(* Call ST08_404_Y52_0 Hub Bandstrecke STN8 AST (Valve) *)
Analyze         (InputExp:=  TRUE,
                 DoAnalyze:= TRUE );
ST08_404_Y52_0.strAnlayse:=Analyze.OutString;
ST08_404_Y52_0                 (Enable  :=  Analyze.ExpResult,
                                sVisu:=Visu.ST08_404_Y52_0,
                                Reset:=gResetAll,
);
ST08_406_B54_1(ValveObject:= ADR(ST08_404_Y52_0));(*Hub Bandstrecke AST*)
ST08_406_B54_2(ValveObject:= ADR(ST08_404_Y52_0));(*Hub Bandstrecke AST*)

(* Rüstsatz Förderband Vereinzelner (Valve) *)
Analyze         (InputExp:=  TRUE,
                 DoAnalyze:= TRUE );
ST08_412_Y55_0.strAnlayse:=Analyze.OutString;
ST08_412_Y55_0                 (Enable  :=  Analyze.ExpResult,
                                sVisu:=Visu.ST08_412_Y55_0,
                                Reset:=gResetAll,
);

ST08_412_B58_0(ValveObject:= ADR(ST08_412_Y55_0));(*ST08_412_B58_0 Rüstsatz Förderband Vereinzelner eingefahren*)
ST08_412_B58_1(ValveObject:= ADR(ST08_412_Y55_0));(*ST08_412_B58_1 Rüstsatz Förderband Vereinzelner ausgefahren*)

(* Rüstsatz Förderband Stopper (Valve) *)
Analyze         (InputExp:=  TRUE,
                 DoAnalyze:= TRUE );
ST08_412_Y55_2.strAnlayse:=Analyze.OutString;
ST08_412_Y55_2                 (Enable  :=  Analyze.ExpResult,
                                sVisu:=Visu.ST08_412_Y55_2,
                                Reset:=gResetAll,
);

ST08_412_B58_2(ValveObject:= ADR(ST08_412_Y55_2));(*ST08_412_B58_2 Rüstsatz Förderband Stopper eingefahren*)
ST08_412_B58_3(ValveObject:= ADR(ST08_412_Y55_2));(*ST08_412_B58_3 Rüstsatz Förderband Stopper ausgefahren*)
END_PROGRAM

(* POU Stations/ST_00/ST00_SFCs/_CallSFCs, ST *)
PROGRAM _CallSFCs
VAR
	b_init							:BOOL:=FALSE;
	FBSocketCloseAll		:FB_SocketCloseAll;

END_VAR
IF	NOT b_init THEN
		FBSocketCloseAll(bExecute:=TRUE);
		IF	FBSocketCloseAll.bBusy THEN
			b_init:=TRUE;
		END_IF
ELSE
	FBSocketCloseAll(bExecute:=FALSE);
END_IF



ST00_CallSFCs();
ST02_CallSFCs();
ST03_CallSFCs();
ST08_CallSFCs();
END_PROGRAM

(* POU Stations/ST_00/ST00_SFCs/ST00_CallSFCs, ST *)
PROGRAM ST00_CallSFCs
VAR

END_VAR
CallSpecialModeSFCs();

HomePositionSFC();
(*ST00_LoadTInfo();*)
ST02_HomePosition();
ST03_HomePosition();
ST08_HomePosition();
END_PROGRAM

(* POU Stations/ST_02_RT_Tampondrucker/ST02_SFCs/ST02_CallSFCs, ST *)
PROGRAM ST02_CallSFCs

VAR
	fb_ton_wz	:TON;
END_VAR
fb_ton_wz(IN:= TRUE, PT:= t#30s , Q=> , ET=> );

(*Aufrufe nur wenn ein Tampondrucker angeschlossen ist, sonst kommen viele Fehlermeldungt*)
IF	gTypeCode=4991 OR		(*102pol*)
	gTypeCode=312	THEN	(*93pol*)
	ST02_Main();
	ST02_Main.FB_CurrentStepHistorie(st_CurrentStep:=ST02_Main.SFCCurrentStep);
	ST02_AutoStop();
	ST02_CallFBs();
END_IF
(*Sonst werden die Visuelemente nicht mit Texten befüllt*)
IF	ModeSelect.Mode<=MODE_MANUAL AND
	NOT fb_ton_wz.Q THEN
	ST02_CallFBs();
END_IF

	(*Sensopart Kamera initialisieren*)
IF 	NOT MP.ST02.SensopartEthernet THEN
	IF NOT ST02_DT_95_A1.b_ready THEN
		ST02_DT_95_A1.b_init := TRUE;
	ELSE
		ST02_DT_95_A1.b_init := FALSE;
	END_IF
ELSE
	(*Sensopart Kamera Ethernet initialisieren*)
	IF NOT ST02_DT_95_A2.st_ctrl_out.b_bereit AND MP.ST02.SensopartIPAdress <>''  THEN
		ST02_DT_95_A2.st_ctrl_in.b_init := TRUE;
	ELSE
		ST02_DT_95_A2.st_ctrl_in.b_init := FALSE;
	END_IF
END_IF
END_PROGRAM

(* POU Stations/ST_02_RT_Tampondrucker/ST02_FBs/ST02_CallFBs, ST *)
PROGRAM ST02_CallFBs
VAR

END_VAR
(*----------------------------------------------------------------------------------------------------------------------------------*)
(* ----------------------------------------------------------------------------------------- *)
(* Call ST02_FDB_40_B61 Iso von SPM auf Band abgelegt (DigIn) *)
ST02_FDB_40_B61                (sVisu:=Visu.ST02_FDB_40_B61,
                                Reset:=gResetAll,
			(*	CheckSignalHigh:=TRUE,*)
);
(* Call ST02_FDB_40_B71 ST02 Iso auf Band vor Vereinzler (DigIn) *)
ST02_FDB_40_B71                (sVisu:=Visu.ST02_FDB_40_B71,
                                Reset:=gResetAll,
			(*	CheckSignalHigh:=TRUE,*)
);
(* Call ST02_S1_6A01 ST02 Sicherung 24V (DigIn) *)
ST02_S1_6A01                (sVisu:=Visu.ST02_S1_6A01,
                                Reset:=gResetAll,
				CheckSignalHigh:=TRUE,
);

(*Sensopart Kamera für die Erkennung der Markierungen*)
ST02_DT_95_A1(
	b_kamera_aktiv:=MP.ST02.CamOn AND NOT MP.ST02.SensopartEthernet,
	st_Description:= 'Kamera Farberkennung',
	b_reset:=gResetAll );

(*Sensopart Kamera für die Erkennung der Markierungen*)
ST02_DT_95_A2(
	st_ctrl_in := ST02_DT_95_A2.st_ctrl_in,
	Activated := MP.ST02.CamOn AND MP.ST02.SensopartEthernet AND MP.ST02.SensopartIPAdress <> '',
	st_Description:= 'Kamera Farberkennung',
	);
IF 	MP.ST02.SensopartIPAdress <> ''  THEN
	ST02_DT_95_A2.s_IpAdress := MP.ST02.SensopartIPAdress;  		(* 'MP.SensopartIPAdress';*)
	ST02_DT_95_A2.i_CmdPort := 2006;
	ST02_DT_95_A2.i_DataPort :=2005;
END_IF

(* Call ST02_S1_70K61_A1 Start  Bedrucken (DigOutIn) *)
ST02_S1_70K61_A1                  (sVisu:=Visu.ST02_S1_70K61_A1,
                                Reset:=gResetAll,
);

(* Call ST02_62_Y6 Tisch drehen 0 - 180 Grad  (Valve) *)
Analyze         (InputExp:=  TRUE,
                 DoAnalyze:= TRUE );
ST02_62_Y6.strAnlayse:=Analyze.OutString;
ST02_62_Y6                 (Enable  :=  Analyze.ExpResult,
                                sVisu:=Visu.ST02_62_Y6,
                                Reset:=gResetAll,
);
ST02_DT_62_B81(ValveObject:= ADR(ST02_62_Y6));(*Tisch drehen 0 Grad*)
ST02_DT_62_B91(ValveObject:= ADR(ST02_62_Y6));(*Tisch drehen 180 Grad*)

IF	ST02_DT_62_B81.ValveSensor THEN
	MP.ST02.TableData[1].ProcessData.Nest_Nr:=2;
	MP.ST02.TableData[2].ProcessData.Nest_Nr:=1;
ELSIF	ST02_DT_62_B91.ValveSensor THEN
	MP.ST02.TableData[1].ProcessData.Nest_Nr:=1;
	MP.ST02.TableData[2].ProcessData.Nest_Nr:=2;
ELSE
	MP.ST02.TableData[1].ProcessData.Nest_Nr:=0;
	MP.ST02.TableData[2].ProcessData.Nest_Nr:=0;
END_IF
(*----------------------------------------------------------------------------------------------------------------------------------*)
(* Call ST02_62_Y9 Schwenkarm 2 drehen 90 - 180 Grad  (Valve) *)
Analyze         (InputExp:=  TRUE,
                 DoAnalyze:= TRUE );
ST02_62_Y9.strAnlayse:=Analyze.OutString;
ST02_62_Y9                 (Enable  :=  Analyze.ExpResult,
                                sVisu:=Visu.ST02_62_Y9,
                                Reset:=gResetAll,
);
(*ST02_DT_61_B21(ValveObject:= ADR(ST02_62_Y9));		(*Schwenkarm 2 90 Grad*)*)
ST02_DT_61_B11(ValveObject:= ADR(ST02_62_Y9));		(*Schwenkarm 2 180 Grad*)

(* Call ST02_62_Y11 Schwenkarm 2 drehen 90 - 0 Grad  (Valve) *)
Analyze         (InputExp:=  TRUE,
                 DoAnalyze:= TRUE );
ST02_62_Y11.strAnlayse:=Analyze.OutString;
ST02_62_Y11                 (Enable  :=  Analyze.ExpResult,
                                sVisu:=Visu.ST02_62_Y11,
                                Reset:=gResetAll,
);
(*ST02_DT_61_B21_clone(ValveObject:= ADR(ST02_62_Y11));(*Schwenkarm 2 90 Grad*)*)
ST02_DT_61_B31(ValveObject:= ADR(ST02_62_Y11));		(*Schwenkarm 2 0 Grad*)


ST02_Schwenkarm[2](
	ST02_90_180:=ST02_62_Y9 ,
	ST02_90_0:=ST02_62_Y11 ,
	ST02_90:=ST02_DT_61_B21);
(*----------------------------------------------------------------------------------------------------------------------------------*)
(* Call ST02_62_Y13 Schwenkarm 1 drehen 90 - 180 Grad  (Valve) *)
Analyze         (InputExp:=  TRUE,
                 DoAnalyze:= TRUE );
ST02_62_Y13.strAnlayse:=Analyze.OutString;
ST02_62_Y13                 (Enable  :=  Analyze.ExpResult,
                                sVisu:=Visu.ST02_62_Y13,
                                Reset:=gResetAll,
);
(*ST02_DT_61_B51(ValveObject:= ADR(ST02_62_Y13));		(*Schwenkarm 1 90 Grad*)*)
ST02_DT_61_B41(ValveObject:= ADR(ST02_62_Y13));		(*Schwenkarm 1 180 Grad*)

(* Call ST02_62_Y15 Schwenkarm 1 drehen 90 - 0 Grad  (Valve) *)
Analyze         (InputExp:=  TRUE,
                 DoAnalyze:= TRUE );
ST02_62_Y15.strAnlayse:=Analyze.OutString;
ST02_62_Y15                 (Enable  :=  Analyze.ExpResult,
                                sVisu:=Visu.ST02_62_Y15,
                                Reset:=gResetAll,
);
(*ST02_DT_61_B51_clone(ValveObject:= ADR(ST02_62_Y15));(*Schwenkarm 1 90 Grad*)*)
ST02_DT_62_B11(ValveObject:= ADR(ST02_62_Y15));		(*Schwenkarm 1 0 Grad*)

ST02_Schwenkarm[1](
	ST02_90_180:=ST02_62_Y13 ,
	ST02_90_0:=ST02_62_Y15,
	ST02_90:=ST02_DT_61_B51);

(* Call ST02_S1_40K01  Freigabe Förderband von SPM (DigIn) *)
ST02_S1_40K01                     (sVisu:=Visu.ST02_S1_40K01,
                                Reset:=gResetAll,
																CheckSignalHigh:=FALSE,
);
(* Call ST02_FDB_80_B02 Band Entnahmeposition 2 (DigIn) *)
ST02_FDB_80_B02                     (sVisu:=Visu.ST02_FDB_80_B02,
                                Reset:=gResetAll
);

(* Call ST02_FDB_54_B41 Kamera ISK anwesend an Prüfposition (DigIn) *)
ST02_FDB_54_B41               (sVisu:=Visu.ST02_FDB_54_B41,
                                Reset:=gResetAll,
);

(* Call ST02_DT_65B11 Tampondrucker Nest 1 leer (DigIn) *)
ST02_DT_65B11               (sVisu:=Visu.ST02_DT_65B11,
                                Reset:=gResetAll,
);

(* Call ST02_DT_65B21 Tampondrucker Nest 2 leer (DigIn) *)
ST02_DT_65B21               (sVisu:=Visu.ST02_DT_65B21,
                                Reset:=gResetAll,
);
(* Init ST02_35_S31 ST02 Druckschalter Wartungseinheit Hauptluft min.6 bar (DigIn) *)
ST02_35_S31 	                (sVisu:=Visu.ST02_35_S31,
                                Reset:=gResetAll,
			CheckSignalHigh:=TRUE,
);
(*----------------------------------------------------------------------------------------------------------------------------------*)
(* Call ST02_FDB_55X1_5_READY IFM Kamera Flügelerkennung links Ready (DigIn) *)
ST02_FDB_55X1_5_READY               (sVisu:=Visu.ST02_FDB_55X1_5_READY,
                                Reset:=gResetAll,
);
(* Call ST02_FDB_55X1_6_IO IFM Kamera Flügelerkennung links Ergebnis iO (DigIn) *)
ST02_FDB_55X1_6_IO               (sVisu:=Visu.ST02_FDB_55X1_6_IO,
                                Reset:=gResetAll,
);
(* Call ST02_FDB_55X1_6_NIO IFM Kamera Flügelerkennung links Ergebnis niO (DigIn) *)
ST02_FDB_55X1_6_NIO               (sVisu:=Visu.ST02_FDB_55X1_6_NIO,
                                Reset:=gResetAll,
);
(* Call ST02_FDB_55X1_2_TRIGGER IFM Kamera Flügelerkennung links Trigger (DigOutIn) *)
ST02_FDB_55X1_2_TRIGGER                  (sVisu:=Visu.ST02_FDB_55X1_2_TRIGGER,
                                Reset:=gResetAll,
);
(* Call ST02_FDB_55X1_7_JOB_BIT1 IFM Kamera  links Jobwechsel Bit1 (DigOutIn) *)
ST02_FDB_55X1_7_JOB_BIT1                  (sVisu:=Visu.ST02_FDB_55X1_7_JOB_BIT1,
                                Reset:=gResetAll,
);
(* Call ST02_FDB_55X1_7_JOB_BIT2 IFM Kamera  links Jobwechsel Bit2 (DigOutIn) *)
ST02_FDB_55X1_7_JOB_BIT2                  (sVisu:=Visu.ST02_FDB_55X1_7_JOB_BIT2,
                                Reset:=gResetAll,
);
(* Call ST02_FDB_56X1_5_READY IFM Kamera Flügelerkennung rechts Ready (DigIn) *)
ST02_FDB_56X1_5_READY               (sVisu:=Visu.ST02_FDB_56X1_5_READY,
                                Reset:=gResetAll,
);
(* Call ST02_FDB_56X1_6_IO IFM Kamera Flügelerkennung rechts Ergebnis iO (DigIn) *)
ST02_FDB_56X1_6_IO               (sVisu:=Visu.ST02_FDB_56X1_6_IO,
                                Reset:=gResetAll,
);
(* Call ST02_FDB_56X1_6_NIO IFM Kamera Flügelerkennung rechts Ergebnis niO (DigIn) *)
ST02_FDB_56X1_6_NIO               (sVisu:=Visu.ST02_FDB_56X1_6_NIO,
                                Reset:=gResetAll,
);
(* Call ST02_FDB_56X1_2_TRIGGER IFM Kamera Flügelerkennung rechts Trigger (DigOutIn) *)
ST02_FDB_56X1_2_TRIGGER                  (sVisu:=Visu.ST02_FDB_56X1_2_TRIGGER,
                                Reset:=gResetAll,
);
(* Call ST02_FDB_56X1_7_JOB_BIT1 IFM Kamera  rechts Jobwechsel Bit1 (DigOutIn) *)
ST02_FDB_56X1_7_JOB_BIT1                  (sVisu:=Visu.ST02_FDB_56X1_7_JOB_BIT1,
                                Reset:=gResetAll,
);
(* Call ST02_FDB_56X1_7_JOB_BIT2 IFM Kamera  rechts Jobwechsel Bit2 (DigOutIn) *)
ST02_FDB_56X1_7_JOB_BIT2                  (sVisu:=Visu.ST02_FDB_56X1_7_JOB_BIT2,
                                Reset:=gResetAll,
);
(* Call ST02_62_Y4 Kamera Ausschleusen Bandstrecke (Valve) *)
Analyze         (InputExp:=  TRUE,
                 DoAnalyze:= TRUE );
ST02_62_Y4.strAnlayse:=Analyze.OutString;
ST02_62_Y4                 (Enable  :=  Analyze.ExpResult,
                                sVisu:=Visu.ST02_62_Y4,
                                Reset:=gResetAll,
);
ST02_FDB_54_B11(ValveObject:= ADR(ST02_62_Y4));(*Kamera Ausschleusen Bandstrecke eingefahren*)
ST02_FDB_54_B21(ValveObject:= ADR(ST02_62_Y4));(*Kamera Ausschleusen Bandstrecke ausgefahren*)


(*Call ST02_62_Y17 Schwenkarm 1 ISK Fixierung ein/ausfahren(Valve) (Valve) *)
Analyze         (InputExp:=  TRUE,
                 DoAnalyze:= TRUE );
ST02_62_Y17.strAnlayse:=Analyze.OutString;
ST02_62_Y17                 (Enable  :=  Analyze.ExpResult,
                                sVisu:=Visu.ST02_62_Y17,
                                Reset:=gResetAll,
);
ST02_S1_66_B11(ValveObject:= ADR(ST02_62_Y17));(*Kamera Ausschleusen Bandstrecke eingefahren*)
ST02_S1_66_B21(ValveObject:= ADR(ST02_62_Y17));(*Kamera Ausschleusen Bandstrecke ausgefahren*)


(*Call ST02_62_Y18 Schwenkarm 2 ISK Fixierung ein/ausfahren(Valve) (Valve) *)
Analyze         (InputExp:=  TRUE,
                 DoAnalyze:= TRUE );
ST02_62_Y18.strAnlayse:=Analyze.OutString;
ST02_62_Y18                 (Enable  :=  Analyze.ExpResult,
                                sVisu:=Visu.ST02_62_Y18,
                                Reset:=gResetAll,
);
ST02_S1_66_B31(ValveObject:= ADR(ST02_62_Y18));(*Kamera Ausschleusen Bandstrecke eingefahren*)
ST02_S1_66_B41(ValveObject:= ADR(ST02_62_Y18));(*Kamera Ausschleusen Bandstrecke ausgefahren*)


(* Call ST02_35Y01 Einschaltventil Hauptluft Tampondruckanlage (Valve) *)
Analyze         (InputExp:=  TRUE,
                 DoAnalyze:= TRUE );
ST02_35Y01.strAnlayse:=Analyze.OutString;
ST02_35Y01               (Enable  :=  Analyze.ExpResult,
                                sVisu:=Visu.ST02_35Y01,
                                Reset:=gResetAll,
);
END_PROGRAM

(* POU Stations/ST_03_Ruestsaetze/ST_03_FBs/ST03_CallSFCs, ST *)
PROGRAM ST03_CallSFCs


VAR


END_VAR
ST03_Main();
ST03_Main.FB_CurrentStepHistorie(st_CurrentStep:=ST03_Main.SFCCurrentStep);


	(*Sensopart Kamera initialisieren*)
IF NOT MP.ST02.SensopartEthernet THEN
	IF NOT ST03_8_80_A1.b_ready THEN
		ST03_8_80_A1.b_init := TRUE;
	ELSE
		ST03_8_80_A1.b_init := FALSE;
	END_IF
	IF NOT ST03_8_85_A1.b_ready THEN
		ST03_8_85_A1.b_init := TRUE;
	ELSE
		ST03_8_85_A1.b_init := FALSE;
	END_IF
ELSE
	(*Sensopart Kamera Ethernet initialisieren*)
	IF NOT ST03_8_90_A1.st_ctrl_out.b_bereit AND MP.ST02.SensopartIPAdress <>''  THEN
		ST03_8_90_A1.st_ctrl_in.b_init := TRUE;
	ELSE
		ST03_8_90_A1.st_ctrl_in.b_init := FALSE;
	END_IF

	IF NOT ST03_8_95_A1.st_ctrl_out.b_bereit AND MP.ST02.SensopartIPAdress2 <>''  THEN
		ST03_8_95_A1.st_ctrl_in.b_init := TRUE;
	ELSE
		ST03_8_95_A1.st_ctrl_in.b_init := FALSE;
	END_IF

	IF NOT ST03_8_100_A1.st_ctrl_out.b_bereit AND MP.ST03.CamOn[1] THEN
		ST03_8_100_A1.st_ctrl_in.b_init := TRUE;
	ELSE
		ST03_8_100_A1.st_ctrl_in.b_init := FALSE;
	END_IF

	IF NOT ST03_8_103_A1.st_ctrl_out.b_bereit AND MP.ST03.CamOn[2] THEN
		ST03_8_103_A1.st_ctrl_in.b_init := TRUE;
	ELSE
		ST03_8_103_A1.st_ctrl_in.b_init := FALSE;
	END_IF

	(*Keyence Kamera Ethernet initialisieren*)
	IF NOT ST03_8_105_A1.st_ctrl_out.b_bereit AND MP.ST03.CamOn_KYE THEN
		ST03_8_105_A1.st_ctrl_in.b_init := TRUE;
	ELSE
		ST03_8_105_A1.st_ctrl_in.b_init := FALSE;
	END_IF


END_IF
END_PROGRAM

(* POU Stations/ST_08_Palettierer/ST_08_SFCs/ST08_CallSFCs, ST *)
 PROGRAM ST08_CallSFCs


VAR


END_VAR
ST08_Process();
ST08_Process.FB_CurrentStepHistorie(st_CurrentStep:=ST08_Process.SFCCurrentStep);

ST08_VV1_Y50_0();
ST08_VV1_Y50_2();

ST08_Depalletizing();
ST08_Depalletizing.FB_CurrentStepHistorie(st_CurrentStep:=ST08_Depalletizing.SFCCurrentStep);

ST08_Palletizing();
ST08_Palletizing.FB_CurrentStepHistorie(st_CurrentStep:=ST08_Palletizing.SFCCurrentStep);
END_PROGRAM

(* POU Stations/ST_08_Palettierer/ST_08_SFCs/Inlett/ST08_VV1_Y50_0, SFC *)
PROGRAM ST08_VV1_Y50_0				(* Vereinzler vor HQE4 *)

VAR_OUTPUT
	SFCCurrentPOU	: STRING:='ST08_VV1_Y50_0';
	SFCCurrentStep	: STRING:='';
	SFCTime			: DINT;
	State   		: DINT;
	Result  		: DINT;
END_VAR
VAR_INPUT

END_VAR
VAR
	MsgOK			: BOOL;
	MsgCancel		: BOOL;
	SFCRun			: BOOL;
	SFCTimeStart	: TIME;
	Delay			: TON;
	TimeOut			: TON;
	(* Userdefinded area *)

END_VAR
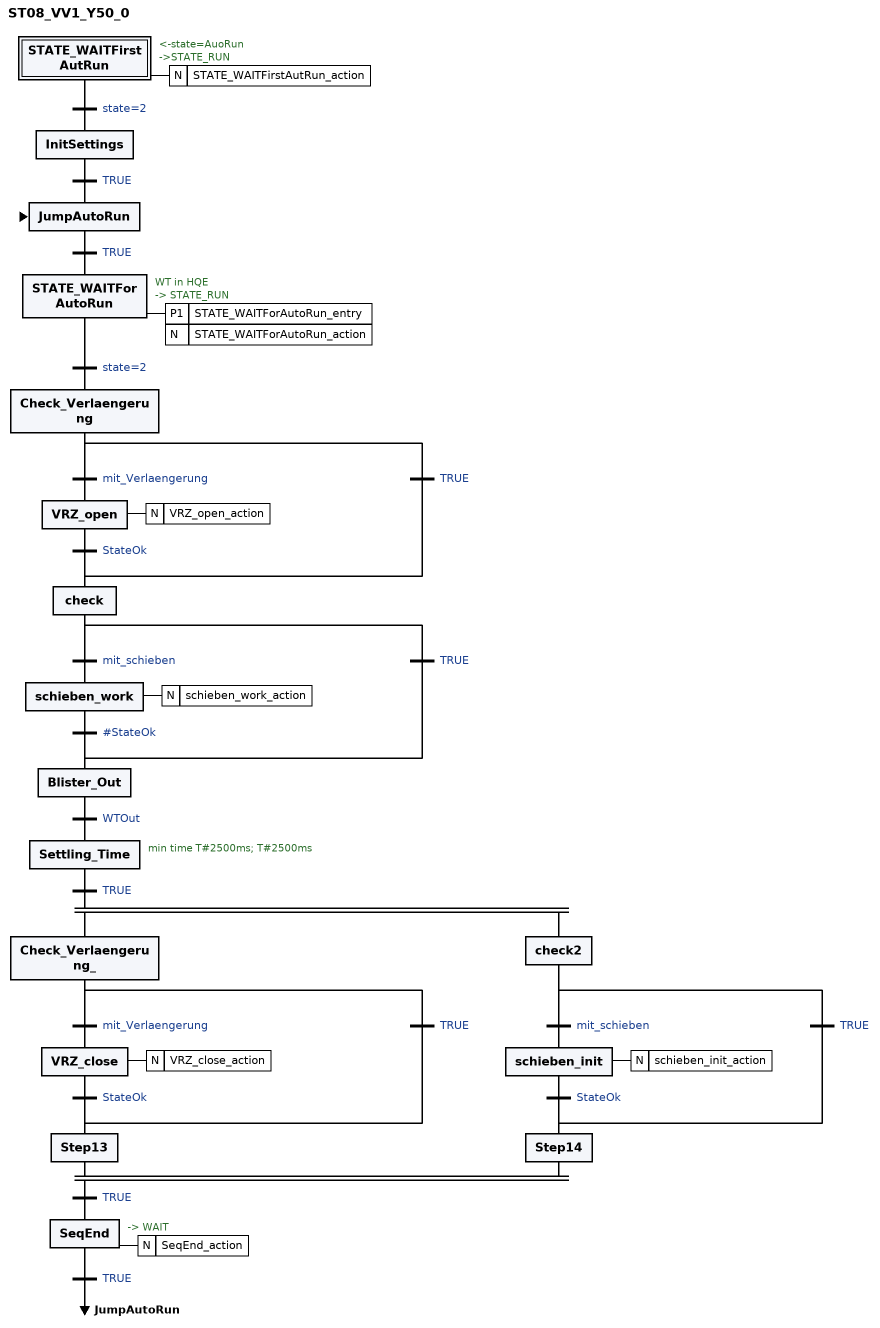
INITIAL_STEP STATE_WAITFirstAutRun: (* <-state=AuoRun / ->STATE_RUN *)
	STATE_WAITFirstAutRun_action(N);
END_STEP
TRANSITION FROM STATE_WAITFirstAutRun TO InitSettings := state=2;
END_TRANSITION
STEP InitSettings:
END_STEP
TRANSITION FROM InitSettings TO JumpAutoRun := TRUE;
END_TRANSITION
STEP JumpAutoRun:
END_STEP
TRANSITION FROM JumpAutoRun TO STATE_WAITForAutoRun := TRUE;
END_TRANSITION
STEP STATE_WAITForAutoRun: (* WT in HQE / -> STATE_RUN *)
	STATE_WAITForAutoRun_entry(P1);
	STATE_WAITForAutoRun_action(N);
END_STEP
TRANSITION FROM STATE_WAITForAutoRun TO Check_Verlaengerung := state=2;
END_TRANSITION
STEP Check_Verlaengerung:
END_STEP
TRANSITION FROM Check_Verlaengerung TO VRZ_open := mit_Verlaengerung;
END_TRANSITION
TRANSITION FROM Check_Verlaengerung TO check := TRUE;
END_TRANSITION
STEP VRZ_open:
	VRZ_open_action(N);
END_STEP
TRANSITION FROM VRZ_open TO check := StateOk;
END_TRANSITION
STEP check:
END_STEP
TRANSITION FROM check TO schieben_work := mit_schieben;
END_TRANSITION
TRANSITION FROM check TO Blister_Out := TRUE;
END_TRANSITION
STEP schieben_work:
	schieben_work_action(N);
END_STEP
TRANSITION FROM schieben_work TO Blister_Out := #StateOk;
END_TRANSITION
STEP Blister_Out:
END_STEP
TRANSITION FROM Blister_Out TO Settling_Time := WTOut;
END_TRANSITION
STEP Settling_Time: (* min time T#2500ms; T#2500ms *)
END_STEP
TRANSITION FROM Settling_Time TO (Check_Verlaengerung_, check2) := TRUE;
END_TRANSITION
STEP Check_Verlaengerung_:
END_STEP
TRANSITION FROM Check_Verlaengerung_ TO VRZ_close := mit_Verlaengerung;
END_TRANSITION
TRANSITION FROM Check_Verlaengerung_ TO Step13 := TRUE;
END_TRANSITION
STEP VRZ_close:
	VRZ_close_action(N);
END_STEP
TRANSITION FROM VRZ_close TO Step13 := StateOk;
END_TRANSITION
STEP Step13:
END_STEP
STEP check2:
END_STEP
TRANSITION FROM check2 TO schieben_init := mit_schieben;
END_TRANSITION
TRANSITION FROM check2 TO Step14 := TRUE;
END_TRANSITION
STEP schieben_init:
	schieben_init_action(N);
END_STEP
TRANSITION FROM schieben_init TO Step14 := StateOk;
END_TRANSITION
STEP Step14:
END_STEP
TRANSITION FROM (Step13, Step14) TO SeqEnd := TRUE;
END_TRANSITION
STEP SeqEnd: (* -> WAIT *)
	SeqEnd_action(N);
END_STEP
TRANSITION FROM SeqEnd TO JumpAutoRun := TRUE;
END_TRANSITION

ACTION STATE_WAITFirstAutRun_action:
IF 		ModeSelect.Mode=MODE_AUTO_RUN
	OR 	ModeSelect.Mode=MODE_STEP_RUN
  OR SpecialMode01.State=State_Run
THEN
	State:=STATE_RUN;
	Result:=RESULT_NON;
ELSE
	State:=STATE_WAIT;
	SFCRun:=FALSE;
(*ELSE*)
END_IF
END_ACTION

ACTION STATE_WAITForAutoRun_entry:
Delay(In:=FALSE);
END_ACTION

ACTION STATE_WAITForAutoRun_action:
Delay(IN:=
	NOT ST08_400_B50_0.BitInToCheck AND
	ST08_401_B50_5.BitInToCheck AND
	ST08_400_Y50_2.InitPosition,
	PT:=T#1500ms);
IF 	((	ModeSelect.Mode=MODE_AUTO_RUN OR 	ModeSelect.Mode=MODE_STEP_RUN   OR SpecialMode01.State=State_Run  )
	AND Delay.Q )

THEN
	State:=STATE_RUN;
	Result:=RESULT_NON;
	SFCTimeStart:=TIME();
ELSE
	State:=STATE_WAIT;
END_IF
END_ACTION

ACTION VRZ_open_action:
ST08_400_Y50_0.MoveWork:=TRUE;
END_ACTION

ACTION schieben_work_action:
ST08_401_Y52_4.MoveWork:=TRUE;
END_ACTION

ACTION VRZ_close_action:
ST08_400_Y50_0.MoveInit:=TRUE;
END_ACTION

ACTION schieben_init_action:
ST08_401_Y52_4.MoveInit:=TRUE;
END_ACTION

ACTION SeqEnd_action:
SFCTime:=TIME_TO_DINT(TIME()-SFCTimeStart);
State:=STATE_WAIT;
END_ACTION

TRANSITION mit_Verlaengerung:
mp.ST08.Trayzufuhr_Verlaengerung
END_TRANSITION

TRANSITION StateOk:
ST08_400_Y50_0.State=STATE_OK
END_TRANSITION

TRANSITION mit_schieben:
MP.ST08.Traystapel_schieben AND
MP.ST08.Trayzufuhr_Verlaengerung
END_TRANSITION

TRANSITION #StateOk:
ST08_401_Y52_4.State=STATE_OK
END_TRANSITION

TRANSITION WTOut:
ST08_400_B50_0.BitInToCheck=TRUE AND ST08_401_B50_5.BitInToCheck=FALSE
END_TRANSITION

TRANSITION mit_Verlaengerung:
MP.ST08.Trayzufuhr_Verlaengerung
END_TRANSITION

TRANSITION StateOk:
ST08_400_Y50_0.State=STATE_OK
END_TRANSITION

TRANSITION mit_schieben:
MP.ST08.Traystapel_schieben AND
MP.ST08.Trayzufuhr_Verlaengerung
END_TRANSITION

TRANSITION StateOk:
ST08_401_Y52_4.State=STATE_OK
END_TRANSITION
END_PROGRAM

(* POU Stations/ST_08_Palettierer/ST_08_SFCs/Inlett/ST08_VV1_Y50_2, SFC *)
PROGRAM ST08_VV1_Y50_2				(* Vereinzler vor HQE4 *)

VAR_OUTPUT
	SFCCurrentPOU	: STRING:='ST08_VV1_Y50_2';
	SFCCurrentStep	: STRING:='';
	SFCTime			: DINT;
	State   		: DINT;
	Result  		: DINT;
END_VAR
VAR_INPUT

END_VAR
VAR
	MsgOK			: BOOL;
	MsgCancel		: BOOL;
	SFCRun			: BOOL;
	SFCTimeStart	: TIME;
	Delay			: TON;
	TimeOut			: TON;
	(* Userdefinded area *)

END_VAR
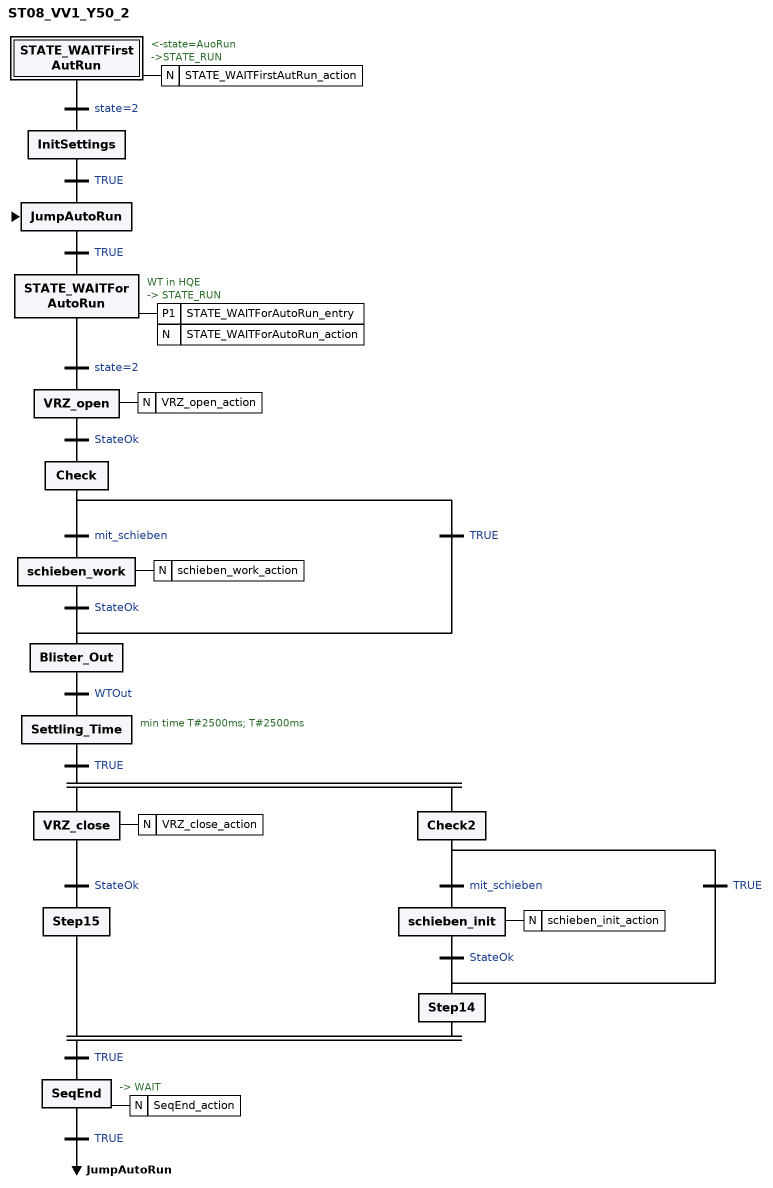
INITIAL_STEP STATE_WAITFirstAutRun: (* <-state=AuoRun / ->STATE_RUN *)
	STATE_WAITFirstAutRun_action(N);
END_STEP
TRANSITION FROM STATE_WAITFirstAutRun TO InitSettings := state=2;
END_TRANSITION
STEP InitSettings:
END_STEP
TRANSITION FROM InitSettings TO JumpAutoRun := TRUE;
END_TRANSITION
STEP JumpAutoRun:
END_STEP
TRANSITION FROM JumpAutoRun TO STATE_WAITForAutoRun := TRUE;
END_TRANSITION
STEP STATE_WAITForAutoRun: (* WT in HQE / -> STATE_RUN *)
	STATE_WAITForAutoRun_entry(P1);
	STATE_WAITForAutoRun_action(N);
END_STEP
TRANSITION FROM STATE_WAITForAutoRun TO VRZ_open := state=2;
END_TRANSITION
STEP VRZ_open:
	VRZ_open_action(N);
END_STEP
TRANSITION FROM VRZ_open TO Check := StateOk;
END_TRANSITION
STEP Check:
END_STEP
TRANSITION FROM Check TO schieben_work := mit_schieben;
END_TRANSITION
TRANSITION FROM Check TO Blister_Out := TRUE;
END_TRANSITION
STEP schieben_work:
	schieben_work_action(N);
END_STEP
TRANSITION FROM schieben_work TO Blister_Out := StateOk;
END_TRANSITION
STEP Blister_Out:
END_STEP
TRANSITION FROM Blister_Out TO Settling_Time := WTOut;
END_TRANSITION
STEP Settling_Time: (* min time T#2500ms; T#2500ms *)
END_STEP
TRANSITION FROM Settling_Time TO (VRZ_close, Check2) := TRUE;
END_TRANSITION
STEP VRZ_close:
	VRZ_close_action(N);
END_STEP
TRANSITION FROM VRZ_close TO Step15 := StateOk;
END_TRANSITION
STEP Step15:
END_STEP
STEP Check2:
END_STEP
TRANSITION FROM Check2 TO schieben_init := mit_schieben;
END_TRANSITION
TRANSITION FROM Check2 TO Step14 := TRUE;
END_TRANSITION
STEP schieben_init:
	schieben_init_action(N);
END_STEP
TRANSITION FROM schieben_init TO Step14 := StateOk;
END_TRANSITION
STEP Step14:
END_STEP
TRANSITION FROM (Step15, Step14) TO SeqEnd := TRUE;
END_TRANSITION
STEP SeqEnd: (* -> WAIT *)
	SeqEnd_action(N);
END_STEP
TRANSITION FROM SeqEnd TO JumpAutoRun := TRUE;
END_TRANSITION

ACTION STATE_WAITFirstAutRun_action:
IF 		ModeSelect.Mode=MODE_AUTO_RUN
	OR 	ModeSelect.Mode=MODE_STEP_RUN
  OR SpecialMode01.State=State_Run
THEN
	State:=STATE_RUN;
	Result:=RESULT_NON;
ELSE
	State:=STATE_WAIT;
	SFCRun:=FALSE;
(*ELSE*)
END_IF
END_ACTION

ACTION STATE_WAITForAutoRun_entry:
Delay(IN:=FALSE);
END_ACTION

ACTION STATE_WAITForAutoRun_action:
Delay(IN:=
	NOT ST08_401_B50_5.BitInToCheck AND
	ST08_402_B51_2.BitInToCheck AND
	ST08_402_Y50_4.InitPosition,
	PT:=T#1500ms);
IF 	((	ModeSelect.Mode=MODE_AUTO_RUN OR 	ModeSelect.Mode=MODE_STEP_RUN   OR SpecialMode01.State=State_Run  )
	AND Delay.Q )

THEN
	State:=STATE_RUN;
	Result:=RESULT_NON;
	SFCTimeStart:=TIME();
ELSE
	State:=STATE_WAIT;
END_IF
END_ACTION

ACTION VRZ_open_action:
ST08_400_Y50_2.MoveWork:=TRUE;
END_ACTION

ACTION schieben_work_action:
ST08_402_Y52_6.MoveWork:=TRUE;
END_ACTION

ACTION VRZ_close_action:
ST08_400_Y50_2.MoveInit:=TRUE;
END_ACTION

ACTION schieben_init_action:
ST08_402_Y52_6.MoveInit:=TRUE;
END_ACTION

ACTION SeqEnd_action:
SFCTime:=TIME_TO_DINT(TIME()-SFCTimeStart);
State:=STATE_WAIT;
END_ACTION

TRANSITION StateOk:
ST08_400_Y50_2.State=STATE_OK
END_TRANSITION

TRANSITION mit_schieben:
MP.ST08.Traystapel_schieben AND
MP.ST08.Trayzufuhr_Verlaengerung
END_TRANSITION

TRANSITION StateOk:
ST08_402_Y52_6.State=STATE_OK
END_TRANSITION

TRANSITION WTOut:
ST08_401_B50_5.BitInToCheck=TRUE AND ST08_402_B51_2.BitInToCheck=FALSE
END_TRANSITION

TRANSITION StateOk:
ST08_400_Y50_2.State=STATE_OK
END_TRANSITION

TRANSITION mit_schieben:
MP.ST08.Traystapel_schieben AND
MP.ST08.Trayzufuhr_Verlaengerung
END_TRANSITION

TRANSITION StateOk:
ST08_402_Y52_6.State=STATE_OK
END_TRANSITION
END_PROGRAM

(* POU Stations/ST_00/ST00_PRGs/_CallPRGs, ST *)
PROGRAM _CallPRGs
VAR
END_VAR
ST00_CallPRGs();
ST02_CallPRGs();
ST03_CallPRGs();
ST08_CallPRGs();
END_PROGRAM

(* POU Stations/ST_00/ST00_PRGs/ST00_CallPRGs, ST *)
PROGRAM ST00_CallPRGs
VAR
	FB_ReadXmlLineConf		: FB_ReadXmlLine;
	sDescription			: STRING;
END_VAR
Lights_and_Lamps();
Safety_Fuses_AirPressure();
JobManagement();
VisuLogger();

IF 	HomePositionSFC.State = STATE_RUN THEN
	ListHomeNOK(InstName:='ST00 ',Description:=sDescription);
END_IF
FB_ReadXmlLineConf(
	Prefix:= 'CONFIG',
	ID:= 'ST00',
	File:= 'CONFIG.xml',
	Text=> sDescription );


IF gInitOk AND ST_Path.Done THEN
	MachineStates();
	ST_Service();
	ST00_ImpExp_MP(
				path:= MP_LocalDriveRoot,
				filename	:=MP_MPExportFilename);
END_IF

(* Schutztüren *)
IF 	ModeSelect.Mode>MODE_MANUAL AND
	ST00_220_S1.BitInToCheck THEN
	ModeSelect.AskForManual:=TRUE;

END_IF

IF	ModeSelect.Mode>MODE_MANUAL THEN
	ST00_220_S1_S31.SetSignalHigh:=TRUE;
	ST00_245_V1.SetSignalHigh:=TRUE;
END_IF

IF 	ModeSelect.Mode<=MODE_MANUAL THEN
	ST00_220_S1_S31.SetSignalLow:=TRUE;
	ST00_245_V1.SetSignalLow:=TRUE;
END_IF

(* Generierung RoboterOffset *)
gRobotOffset :=  TD.RobotOffset;

gTypeCode:=STRING_TO_DINT(DELETE(TD.TypeCode,1,1));
END_PROGRAM

(* POU Stations/ST_00/ST00_PRGs/Lights_and_Lamps, ST *)
PROGRAM Lights_and_Lamps
VAR
	SignalRed			: BOOL;
	SignalOrange		: BOOL;
	SignalGreen			: BOOL;
	SignalBlue			: BOOL;
	SetOrange			: BOOL;
	FP_MachineLight	: R_TRIG;
	FN_MachineLight	: F_TRIG;
	PartLack			: TON;
	TimeOFF			: TON;
	fb_Blinker			: FB_Blinker;
END_VAR
fb_Blinker(b_start:=TRUE, t_taktzeit_on:=t#1s , t_taktzeit_off:=t#1s , b_blinker_out=> );
(* ----------------------------------------------------------------------------------------- *)
(* Ampel  *)
SignalRed	:= ErrorHandler.bOutError ;
SignalOrange	:= MessageHandler.MessageActive OR SetOrange OR ST03_Test_Parts.fb_Blinker.b_blinker_out;;
IF	ModeSelect.Mode=MODE_AUTO_RUN OR ModeSelect.Mode=MODE_STEP_RUN THEN
	SignalGreen	:=TRUE;
ELSIF
	 ModeSelect.Mode=MODE_AUTO_STOP THEN
	SignalGreen	:=fb_Blinker.b_blinker_out;
ELSE
	SignalGreen	:=FALSE;
END_IF
(*SignalGreen	:= ModeSelect.Mode=MODE_AUTO_RUN OR ModeSelect.Mode=MODE_AUTO_STOP OR ModeSelect.Mode=MODE_STEP_RUN;*)
SignalBlue	:= FALSE; (* Parts Missing *)

(* ----------------------------------------------------------------------------------------- *)
PartLack(IN:= FALSE,PT:=T#60s);
IF  	ModeSelect.Mode>MODE_MANUAL AND
	PartLack.Q THEN
	SetOrange:=TRUE;
ELSE
	SetOrange:=FALSE;
END_IF

IF	CurrentVisu <> 'MANUAL_ST00_0' THEN

	(* Ampel Grün *)
	IF 	ST00_350_H1.State=STATE_WAIT AND
		ST00_350_H1.SignalOut <> SignalRed THEN
		ST00_350_H1.SetSignalHigh:= SignalRed;
		ST00_350_H1.SetSignalLow:= NOT SignalRed;
	END_IF;

	(* Ampel Orange *)
	IF 	ST00_350_H2.State=STATE_WAIT AND
		ST00_350_H2.SignalOut <> SignalOrange	THEN
		ST00_350_H2.SetSignalHigh:= SignalOrange;
		ST00_350_H2.SetSignalLow:= NOT SignalOrange;
	END_IF;
	(* Ampel Rot *)
	IF 	ST00_350_H3.State=STATE_WAIT AND
		ST00_350_H3.SignalOut <> SignalGreen THEN
		ST00_350_H3.SetSignalHigh:= SignalGreen;
		ST00_350_H3.SetSignalLow:= NOT SignalGreen;
	END_IF;
	(*Ampel Blau*)
	(*IF 	ST00_350_H4.State=STATE_WAIT AND
		ST00_350_H4.SignalOut <> SignalBlue THEN
		ST00_350_H4.SetSignalHigh:= SignalBlue;
		ST00_350_H4.SetSignalLow:= NOT SignalBlue;
	END_IF*)

(* Bedientaster-Beleuchtungen *)
	(* H3 Reset *)
	IF 	ST00_292_H3_RESET.State=STATE_WAIT AND
		ST00_292_H3_RESET.SignalOut <> SignalRed THEN
		ST00_292_H3_RESET.SetSignalHigh:=SignalRed;
		ST00_292_H3_RESET.SetSignalLow:= NOT SignalRed;
	END_IF;
	(* H2 Start *)
	IF 	ST00_292_H2_Start.State=STATE_WAIT AND
		ST00_292_H2_Start.SignalOut <> SignalGreen 	THEN
		ST00_292_H2_Start.SetSignalHigh:=SignalGreen;
		ST00_292_H2_Start.SetSignalLow:= NOT SignalGreen;
	END_IF

	(* H3 Reset *)
	IF 	ST00_245_V3_RESET.State=STATE_WAIT AND
		ST00_245_V3_RESET.SignalOut <> SignalRed THEN
		ST00_245_V3_RESET.SetSignalHigh:=SignalRed;
		ST00_245_V3_RESET.SetSignalLow:= NOT SignalRed;
	END_IF;
	(* H2 Start *)
	IF 	ST00_245_V2_START.State=STATE_WAIT AND
		ST00_245_V2_START.SignalOut <> SignalGreen 	THEN
		ST00_245_V2_START.SetSignalHigh:=SignalGreen;
		ST00_245_V2_START.SetSignalLow:= NOT SignalGreen;
	END_IF
END_IF

(* Beleuchtung Anlage Ein, wenn Schutz geöffnet*)
(* ----------------------------------------------------------------------------------------- *)

(* Flag Positive - Light on*)
FP_MachineLight(CLK:=NOT gReadyForControlOn );

(* Flag Negative - Light on*)
FN_MachineLight(CLK:=NOT gReadyForControlOn );

TimeOFF(IN:=ST00_31_K1.SignalOut, PT:=t#5m);

IF 	FP_MachineLight.Q THEN
	ST00_31_K1.SetSignalHigh	:= TRUE;
	ST00_31_K1.SetSignalLow	:= FALSE;
END_IF
IF 	FN_MachineLight.Q OR
	TimeOFF.Q THEN
	ST00_31_K1.SetSignalHigh	:= FALSE;
	ST00_31_K1.SetSignalLow	:= TRUE;
END_IF
END_PROGRAM

(* POU zLibrary/ept/Funktionsbausteine/FB_Blinker, ST *)
FUNCTION_BLOCK FB_Blinker
VAR_INPUT
	b_start 		: BOOL;
	t_taktzeit_on	: TIME;
	t_taktzeit_off	: TIME;
END_VAR
VAR_OUTPUT
	b_blinker_out : BOOL;
END_VAR
VAR
	fb_ton		: TON;
END_VAR
fb_ton(IN:=NOT fb_ton.Q AND b_start , PT:=t_taktzeit_off + t_taktzeit_on , Q=> , ET=> );
b_blinker_out:= fb_ton.ET >= t_taktzeit_off;
END_FUNCTION_BLOCK

(* POU Stations/ST_03_Ruestsaetze/ST_03_SFCs/ST03_Test_Parts, ST *)
PROGRAM ST03_Test_Parts
VAR
	FB_Blinker					: FB_Blinker;
END_VAR
(* An der Oberfläche muss bestätigt werden, dass die Prüfteile entnommen worden sind *)
IF 	gTakeTestPartsFinished OR
	ST_CPU.LNG <> CZ THEN
	ST03_Main.TestPartsRemove := FALSE;
END_IF

(* Meldung blinken bis Teile entnommen werden / Blikani okna odeber vzorky do potvrzeni odebrani*)
fb_Blinker(b_start:=ST03_Main.TestPartsRemove , t_taktzeit_on:=t#1s , t_taktzeit_off:=t#1s , b_blinker_out=> );

(*Beim Dummytest 160 polig dürfen die Isos nicht bedruckt werden
	/ Stop Printing at Dummytest 160 pol*)

IF	gTypeCode=322	THEN 	(*160 polig*)
	IF 	NOT DummyTest_160pol THEN
		IF	ST03_8_B76_1.BitInToCheck OR  (* 3621 *)
			ST03_423_B66_0.BitInToCheck THEN (* Rüstsatz 160 polig LS 1 *)
			ST03_PLAN_70V1_1.SetSignalHigh	:= TRUE;		(* Start  Bedrucken Tintenstrahldrucker Frontseite*)
			ST03_PLAN_70V1_1.SetSignalLow	:= FALSE;
		ELSE
			ST03_PLAN_70V1_1.SetSignalHigh	:= FALSE;	(* Start  Bedrucken Tintenstrahldrucker Frontseite*)
			ST03_PLAN_70V1_1.SetSignalLow	:= TRUE;
		END_IF
		IF	ST03_8_B76_2.BitInToCheck OR (* 3621 *)
			ST03_422_B64_0.BitInToCheck THEN  (* Rüstsatz 160 polig LS 2 *)
			ST03_PLAN_71V1_2.SetSignalHigh	:= TRUE;		(* Start  Bedrucken Tintenstrahldrucker Rückseite*)
			ST03_PLAN_71V1_2.SetSignalLow	:= FALSE;
		ELSE
			ST03_PLAN_71V1_2.SetSignalHigh	:= FALSE;	(* Start  Bedrucken Tintenstrahldrucker Rückseite*)
			ST03_PLAN_71V1_2.SetSignalLow	:= TRUE;
		END_IF
	END_IF
END_IF

	(*  Nur in CZ
	Bei erreichen der vorgegebenen Stückzahl werden automatisch Testteile abgelegt
	Spusteni vzorku pri dosazeni zadane hodnoty *)

IF 	ST_CPU.LNG = CZ AND
	NOT MP.ST02.DummyPruefung_93pol THEN
	IF 	gPartsTest >= gPartsTestVisu AND
		NOT gTakeTestPartsAuto	THEN
		gTakeTestPartsAuto:=TRUE;
	END_IF

	IF 	gPartsTest >= gPartsTestVisu THEN
		gPartsTest:=0;
	END_IF
ELSE
	gTakeTestPartsAuto:=FALSE;
	IF 	gTakeTestParts  THEN
		gPartsTest:=0;
	END_IF
END_IF
END_PROGRAM

(* POU Stations/ST_00/ST00_PRGs/JobManagement, ST *)
PROGRAM JobManagement
VAR
	(*Buttons*)
	BtnOffsetPlus				: VisuButton;
	VisuBtnOffsetPlus			: sButtonVisu;
	BtnOffsetMinus				: VisuButton;
	VisuBtnOffsetMinus			: sButtonVisu;
	BtnClearAll					: VisuButton;
	VisuBtnClearAll				: sButtonVisu;
	BtnTestParts				: VisuButton;
	VisuBtnTestParts			: sButtonVisu;

END_VAR
(*Gesamt-IO zuweisen, Gesamt-NIO ermitteln
  ---------------------------------------------------------------------------------*)
MP.ST00.PartsNokTotal:=0;
(*
FOR StIdx:=1 TO NO_OF_NEST
DO
	MP.ST00.PartsNokTotal:=MP.ST00.PartsNokTotal+MP.ST00.PartsNok_ST02[StIdx];
END_FOR
*)
MP.ST00.PartsNokTotal:=0;
MP.ST00.PartsOkTotal:=0;

(*Noch zu produzierende Teile ermitteln
  ---------------------------------------------------------------------------------*)
MP.ST00.PartsRemaining:=(		MP.ST00.PartsToProduce
										 		+ 	MP.ST00.PartsToProduceOffset
										 		- 	gPartsInserted
										 													);

(*Korrekturwert für Sollstückzahl erhöhen bzw verringern
  ---------------------------------------------------------------------------------*)
BtnOffsetPlus(Button:=VisuBtnOffsetPlus,
							Enable:=TRUE,
							Visible:=TRUE,
							TextOn:='+',
							);
BtnOffsetMinus(	Button:=VisuBtnOffsetMinus,
								Enable:=MP.ST00.PartsToProduceOffset>0,
								Visible:=TRUE,
								TextOn:='-');

IF BtnOffsetPlus.PressedFlag THEN
	MP.ST00.PartsToProduceOffset:=MP.ST00.PartsToProduceOffset+1;
END_IF
IF BtnOffsetMinus.PressedFlag THEN
	MP.ST00.PartsToProduceOffset:=MP.ST00.PartsToProduceOffset-1;
END_IF

(*Alle Zähler löschen
  ---------------------------------------------------------------------------------*)
BtnClearAll(Button:=VisuBtnClearAll,
						Enable:=TRUE,
						Visible:=TRUE,
						TextOn:='Alle Zähler löschen',
						);
IF BtnClearAll.PressedFlag THEN
	MP.ST00.PartsToProduce:=0;
	MP.ST00.PartsToProduceOffset:=0;
	MP.ST00.PartsNokSubsetSize:=0;
	gPartsInserted:=0;
	gNokPartsColorCam:=0;
	gNokPartsWingCam:=0;
	gNokPartsPrint:=0;
	NokCounter1li:= 0;
	NokCounter1re:= 0;
	NokCounter2li:= 0;
	NokCounter2re:= 0;
	NokCounter3li:= 0;
	NokCounter3re:= 0;
	i32_first_parts :=0;
END_IF

(*Test Teile entnehmen
  ---------------------------------------------------------------------------------*)
BtnTestParts(	Button:=VisuBtnTestParts,
						Enable:=TRUE,
						Visible:=ModeSelect.Mode=MODE_AUTO_RUN AND
								NOT ST03_Main.TestPartsRemove,
						TextOn:='TestParts',
				);

IF 	ModeSelect.Mode=MODE_AUTO_RUN AND BtnTestParts.PressedFlag THEN
  	gTakeTestParts:=TRUE;
ELSIF
	ModeSelect.Mode<>MODE_AUTO_RUN THEN
	gTakeTestParts:=FALSE;
END_IF
END_PROGRAM

(* POU Stations/ST_00/ST00_PRGs/VisuLogger, ST *)
PROGRAM VisuLogger
VAR
	PageHistory		: ARRAY[1..20] OF STRING(40);
	Trigger				: BOOL;
	Clock					: R_TRIG;
	LastVisuPage	: STRING(40);
	bDeleteBuf		: BOOL;
	i							: INT;
END_VAR
IF 	LastVisuPage='' THEN
	LastVisuPage:=CurrentVisu;
END_IF

Trigger:=CurrentVisu<>LastVisuPage;
Clock(Clk:=Trigger);

IF 	Clock.Q THEN
	FOR i:= 20 TO 2 BY -1 DO
		PageHistory[i]:=PageHistory[i-1];
	END_FOR
	PageHistory[1]:=CurrentVisu;
END_IF

IF 	bDeleteBuf THEN
	FW_MemSet(ADR(PageHistory), 0, SIZEOF(PageHistory));
	bDeleteBuf:=FALSE;
END_IF

LastVisuPage:=CurrentVisu;
END_PROGRAM

(* POU Stations/ST_00/ST00_PRGs/MachineStates, ST *)
PROGRAM MachineStates
VAR
	InfoNoUser				: ErrorStruct;
	LogFileEntry			: ErrorStruct;
	FP_AutoRun				: R_TRIG;
	FirstCycle				: BOOL := TRUE;
	FP_STOP					: R_TRIG;
	TON_STOP				: TON;
	CycleTime             	: REAL;
	CycleTimeHelp           : STRING;

	FB_ReadXmlLineMsg		: FB_ReadXmlLine;
	FB_ReadXmlLineUser		: FB_ReadXmlLine;

	s_MsgNew				: STRING;
	s_UserNew				: STRING;
END_VAR
(* Programmaufrufe *)
_Message();

(*Open Main-Screen with AutoStart-Button*)
FP_AutoRun(CLK:= ModeSelect.Mode=MODE_AUTO);

IF FP_AutoRun.Q THEN
	CurrentVisu:='MAIN';
END_IF

(* SYSTEM_GST *)
IF ModeSelect.HomePosRunFirstImp THEN
	CurrentVisu:='SYSTEM_GST';
END_IF


(*Button "Leerfahren" einblenden*)
ModeSelect.ShowBtnRunEmpty:=TRUE;

(*Taster "Start" und "Stop" am Schaltschrank*)
IF 	(ModeSelect.Mode<=MODE_MANUAL AND ModeSelect.BtnManual.Visible OR ModeSelect.Mode=MODE_AUTO)AND
	(ST00_292_S2_START.BitInToCheck OR ST00_245_S2_START.BitInToCheck) THEN
	ModeSelect.iRemoteAutoStart:=TRUE;
END_IF

FP_STOP(CLK:=ST00_292_S1_STOP.BitInToCheck OR ST00_245_S1_STOP.BitInToCheck);

IF 	ModeSelect.Mode=MODE_AUTO_RUN AND
	FP_STOP.Q THEN
	ModeSelect.iRemoteAutoStop:=TRUE;
END_IF

IF 	ModeSelect.Mode=MODE_AUTO AND
	FP_STOP.Q THEN
	ModeSelect.AskForManual:=TRUE;
END_IF


CycleTime:=DINT_TO_REAL (ST03_Main.SFCTime);

CycleTime:=(CycleTime/10000);
CycleTimeHelp:=REAL_TO_STRING(CycleTime);
CycleTimeHelp:=LEFT(CycleTimeHelp,4);

(* Force ManualMode if AutoStop not successful *)
TON_STOP(IN:=ST00_292_S1_STOP.SignalIn OR ST00_245_S1_STOP.SignalIn, PT:=t#1s );
IF 	ModeSelect.Mode=MODE_AUTO_STOP AND
	TON_STOP.Q THEN
	ModeSelect.AskForManual:=TRUE;
END_IF

(*Force HomePosition-Run after every Manual-Mode*)
IF 	ModeSelect.Mode<=MODE_MANUAL THEN
	gHomePosSFCDone:=FALSE;
END_IF

IF 	ModeSelect.Mode<>MODE_Special THEN
	DummyTest_160pol := FALSE;
	MP.ST02.DummyPruefung_93pol :=FALSE;
END_IF
END_PROGRAM
ACTION _Message:
(* setze Dateinamen für Fehlerdatei *)
ErrorHandler.ErrorLogFileName := CONCAT(LOG_RDPathLocal,'ErrorLog_');
ErrorHandler.ErrorLogFileName := CONCAT(ErrorHandler.ErrorLogFileName, WORD_TO_STRING(CallGeneralFunctions.wYear));
ErrorHandler.ErrorLogFileName := CONCAT(ErrorHandler.ErrorLogFileName, '-');
ErrorHandler.ErrorLogFileName := CONCAT(ErrorHandler.ErrorLogFileName, WORD_TO_STRING(CallGeneralFunctions.wMonth));
ErrorHandler.ErrorLogFileName := CONCAT(ErrorHandler.ErrorLogFileName, '.csv');



(*LogFile-Eintrag bei Betriebsarten-Umschaltung*)
IF 	FirstCycle THEN
	FB_ReadXmlLineMsg.ID:='bm_restart';
	FirstCycle:=FALSE;
ELSIF
	ModeSelect.ManualFirstImp THEN
	FB_ReadXmlLineMsg.ID:='bm_manual_mode';
ELSIF
	ModeSelect.AutoFirstImp THEN
	FB_ReadXmlLineMsg.ID:='bm_automatic_mode';
ELSIF
	ModeSelect.HomePosRunFirstImp THEN
	FB_ReadXmlLineMsg.ID:='bm_homepos';
END_IF

IF	s_MsgNew <> FB_ReadXmlLineMsg.Text AND
	FB_ReadXmlLineMsg.Text <> '' THEN
	LogFileEntry.DateTime:=gVarDTSystemtime;
	LogFileEntry.Text  	:=FB_ReadXmlLineMsg.Text;
	LogFileEntry.Typ   	:=1; (*yellow Info-Line*)
	LogFileEntry.No    	:=1;
	ErrorHandler.AddError(ErrorToAdd:=LogFileEntry,sVisu:=Visu.ErrorHandler);
	s_MsgNew:=FB_ReadXmlLineMsg.Text;
END_IF



(*Show a Message when no User is logged in*)
IF	NOT UserLoginHandler.UserLoggedIn THEN
	FB_ReadXmlLineUser.ID:='bm_user_not_login';
END_IF

IF	s_UserNew <> FB_ReadXmlLineUser.Text AND
	FB_ReadXmlLineUser.Text <> '' THEN
	InfoNoUser.DateTime:=gVarDTSystemtime;
	InfoNoUser.Text  	:=FB_ReadXmlLineUser.Text;
	InfoNoUser.Typ   	:=2; (*yellow Info-Line*)
	InfoNoUser.No    	:=1;
	ErrorHandler.AddError(ErrorToAdd:=InfoNoUser,sVisu:=Visu.ErrorHandler);
	s_UserNew:=FB_ReadXmlLineUser.Text;
END_IF



(*Aufrufe*)
FB_ReadXmlLineMsg(
	Prefix:= 'MSG',
	File:= 'MSG.xml');

FB_ReadXmlLineUser(
	Prefix:= 'MSG',
	File:= 'MSG.xml');
END_ACTION

(* POU zLibrary/ept/Service/ST_Service, ST *)
PROGRAM ST_Service
VAR_INPUT
	st_ctrl_in						: struct_ctrl_in;
END_VAR
VAR_OUTPUT
	Error							:BOOL;
	ErrorMsg: STRING(255);	(*  *)
	ErrorID					:STRING(20);
END_VAR
VAR
	b_first_cycle					: BOOL := TRUE;
	fb_state_entry				: ST_StateEntry;

	fb_ton_uez						: TON;
	fb_ton_wz									: TON;
	fb_r_trig_counter					:R_TRIG;
	i_aktueller_tag						: INT;
	lr_aktuelle_stunden				: LREAL;
	i_aktuelle_stunden				: INT;
	MsgOK											:BOOL;
	fb_bbgen_xml_file					: ST_BBGenXMLFile;
	Service_daten_copy				: ARRAY [0..15] OF struct_daten_service;
	betriebssekundenzaehler_copy	:UDINT;
	M_BtnType									: ARRAY[0..15] OF BOOL;
	HelpString						:STRING(255);
	FB_Betriebsstundenzaehler	:FB_Betriebsstundenzaehler;
	lr_Betriebsstunden					:LREAL;
	Start								:BOOL;
	gPartsInsertedCopy				: DINT;
	i_act_ErrorNumber				:INT;
	ColorName							: ARRAY[0..15] OF DINT; (*from STRUCT Colors*)
	Default_reached						: ARRAY[0..15] OF BOOL; 	 (*Merker damit Fehlermeldung nur einmal angezeigt wird*)
	Warning_reached						: ARRAY[0..15] OF BOOL;	(*Merker damit Warnmeldung nur einmal angezeigt wird*)
	Reset_Help						: ARRAY[1..3] OF BOOL;

	CURRENTLANGUAGECopy			: STRING(5);

	fb_ExpActService				: FB_ExporString;	(* Fehlermeldungen in Errorlog (txt) schreiben *)
END_VAR
VAR_TEMP
	i					:INT:=-1;
	k					:INT:=-1;
END_VAR
Reset();

FB_Betriebsstundenzaehler(
	Start:= ModeSelect.Mode=MODE_AUTO_RUN OR Start,
	Reset:= ,
	i32_betriebssekundenzaehler_in:= Service.betriebssekundenzaehler,
	i32_betriebssekundenzaehler=> Service.betriebssekundenzaehler,
	lr_betriebsstundenzaehler=> lr_Betriebsstunden);

(*Zeiten*)
fb_ton_uez(IN:= , PT:= , Q=> , ET=> );
fb_ton_wz(IN:= , PT:= , Q=> , ET=> );

(*Flanken*)
fb_r_trig_counter(CLK:= gPartsInsertedCopy<>gPartsInserted, Q=> );	(*ST02_160_A1_3.BitOutToSet	 Signal von Rundschalttisch drehen *)
gPartsInsertedCopy:=gPartsInserted;

(* Hochzählen der einelnen Zähler *)
IF fb_r_trig_counter.Q THEN
	FOR i:=0 TO 15 BY 1 DO
		IF Service.daten[i].Type_Service = COUNTER AND Service.daten[i].Default_Value > 0 THEN
			Service.daten[i].Current_Value := Service.daten[i].Current_Value +1;
		END_IF
	END_FOR
END_IF

(* Tage seit dem 01.01.2000 *)
i_aktueller_tag := (WORD_TO_INT (gVarSystemtime.wYear) - 2000) *360;	(* Anzahl der Jahre x360 Tage *)
i_aktueller_tag := i_aktueller_tag + (WORD_TO_INT (gVarSystemtime.wMonth)*30) ;	(* Anzahl der Monate x30 Tage *)
i_aktueller_tag := i_aktueller_tag + WORD_TO_INT (gVarSystemtime.wDay);	(* Anzahl der Tage *)

lr_aktuelle_stunden:=WORD_TO_LREAL(gVarSystemtime.wHour)+
										(WORD_TO_LREAL(gVarSystemtime.wMinute)/60);		(*Anzahl der Stunden*)
i_aktuelle_stunden:=LREAL_TO_INT(lr_aktuelle_stunden*100);
lr_aktuelle_stunden:=INT_TO_LREAL(i_aktuelle_stunden)/100;


Umschalten();

(*===================================================================================================================================*)

(* Toplevel *)
IF fb_state_entry.i16_next_step > INIT AND fb_state_entry.i16_next_step < FEHLER THEN
	IF fb_state_entry.i16_next_step < STOP THEN
		IF st_ctrl_in.b_stop THEN
			fb_state_entry.i16_next_step := STOP;
		END_IF
	END_IF
END_IF


fb_state_entry(i16_pos:= 1);

CASE fb_state_entry.i16_step OF
(*=======================================================*)
	INIT_OBJ:

		IF 	b_first_cycle THEN	(* Programmstart >> XML Datei auslesen *)
			fb_state_entry.i16_next_step := 200;
		ELSE
			fb_state_entry.i16_next_step := INIT;
		END_IF

(*=======================================================*)
	INIT:
		IF fb_state_entry.E THEN
			i := -1;
			Error := FALSE;
			fb_bbgen_xml_file.start_lesen_service := FALSE;
			fb_bbgen_xml_file.start_schreiben_service := FALSE;
			FOR i:=0 TO 15 BY 1 DO
				ColorName[i]:=color.white;
				Service.daten[i].Warning_reached := FALSE;
				Service.daten[i].Default_reached := FALSE;
			END_FOR
		END_IF

		(*-----------------------Weiterschaltbedingungen----------------------------*)
		IF NOT fb_state_entry.E THEN
			fb_state_entry.i16_next_step := BEREIT;
		END_IF

(*=======================================================*)
	BEREIT:		fb_state_entry.s_debugtext:='warte auf Änderung oder Sprachumschaltung';

		IF 	fb_state_entry.E AND i_act_ErrorNumber<> -1THEN
			ColorName[i_act_ErrorNumber]:=color.white;
			i_act_ErrorNumber:=-1;
		END_IF

		(*-----------------------Weiterschaltbedingungen----------------------------*)
		i := -1;
		FOR i:=0 TO 15 BY 1 DO

		(* Wenn Vorgabewert erreicht wird und der Start Button betätigt wird, wird eine Meldung ausgegeben *)
			IF 	Service.daten[i].Default_reached AND
				i_act_ErrorNumber =-1 AND
				NOT Default_reached[i]  THEN

					ErrorMsg:= CONCAT (Service.daten[i].Name, ' Vorgabewert erreicht');
					Default_reached[i]:=TRUE;
					i_act_ErrorNumber:=i;
					ColorName[i]:=color.lightgrey;
					fb_state_entry.i16_next_step:=FEHLER;

			END_IF

		(* Wenn Warngrenze erreicht wird und der Start Button betätigt wird, wird eine Meldung ausgegeben *)
			IF 	Service.daten[i].Warning_reached  AND
				i_act_ErrorNumber =-1 AND
				NOT Service.daten[i].Default_reached AND
				NOT Warning_reached[i] THEN

					Warning_reached[i]:=TRUE;
					i_act_ErrorNumber:=i;
					ErrorID:='';
					ErrorMsg:= CONCAT (Service.daten[i].Name, ' Warngrenze erreicht');
					ColorName[i]:=color.lightgrey;
					fb_state_entry.i16_next_step:=STOP;

			END_IF
		END_FOR

		IF	CURRENTLANGUAGECopy <> CURRENTLANGUAGE THEN
			fb_state_entry.i16_next_step := 200;
		END_IF

		(* Wenn Unterschied und im Handbetrieb, dann schreibe XML *)
		IF 	(MEMCMP(ADR(Service_daten_copy), ADR(Service.daten), SIZEOF(Service_daten_copy)) <> 0 ) AND
			(ModeSelect.Mode = MODE_MANUAL OR ModeSelect.Mode = MODE_NON) OR
			betriebssekundenzaehler_copy <> service.betriebssekundenzaehler THEN
			fb_bbgen_xml_file.start_lesen_service := FALSE;
			fb_bbgen_xml_file.start_schreiben_service := FALSE;
			fb_state_entry.i16_next_step:=110;
		END_IF

(*=======================================================*)
	110:	fb_state_entry.s_debugtext:='XML Schreiben';

		IF fb_state_entry.E THEN
			fb_bbgen_xml_file.start_schreiben_service := TRUE;
			fb_bbgen_xml_file.s_path := MP_TDPathService;
			fb_bbgen_xml_file.s_service := CONCAT(CURRENTLANGUAGE,'_Service');
		END_IF

		(*-----------------------Weiterschaltbedingungen----------------------------*)
		IF fb_bbgen_xml_file.fertig_schreiben AND NOT fb_state_entry.E THEN
			fb_bbgen_xml_file.start_schreiben_service := FALSE;
			Service_daten_copy := Service.daten;
			betriebssekundenzaehler_copy:=service.betriebssekundenzaehler;
			fb_state_entry.i16_next_step := BEREIT;
		ELSIF fb_bbgen_xml_file.bError THEN
			ErrorID:='PM1';
			ErrorMsg:= ' Fehler beim Schreiben der Service XML-Datei';
			fb_state_entry.i16_next_step := FEHLER;
		END_IF

(*=======================================================*)
	200:	fb_state_entry.s_debugtext:=CONCAT(CURRENTLANGUAGE,'_Servie.xml einlesen');

		IF fb_state_entry.E THEN
			fb_bbgen_xml_file.start_lesen_service := TRUE;
			fb_bbgen_xml_file.s_path := MP_TDPathService;
			fb_bbgen_xml_file.s_service := CONCAT(CURRENTLANGUAGE,'_Service');
			fb_ExpActService.Start:=TRUE;
		END_IF

		(*-----------------------Weiterschaltbedingungen----------------------------*)
		IF fb_bbgen_xml_file.fertig_lesen AND NOT fb_state_entry.E THEN
			CURRENTLANGUAGECopy:=CURRENTLANGUAGE;
			fb_bbgen_xml_file.start_lesen_service := FALSE;
			Service_daten_copy := Service.daten;
			betriebssekundenzaehler_copy:=service.betriebssekundenzaehler;
			Button_Init();
			b_first_cycle := FALSE;
			fb_state_entry.i16_next_step := INIT;
		ELSIF
			fb_bbgen_xml_file.bError OR fb_bbgen_xml_file.nErrId  <> 0 THEN
			ErrorID:='PM2';
			ErrorMsg:= '';
			ErrorMsg:= ' Fehler beim Lesen der Service XML-Datei';
			fb_state_entry.i16_next_step := FEHLER;
		END_IF

(*=======================================================*)
	FEHLER:
		IF fb_state_entry.E THEN
			MessageHandler.ClearMessageLines(sVisu:=Visu.Message);
		END_IF
		MessageHandler.Msg.ID:=ErrorID;
		MessageHandler.Msg.Color:=Color.red;
		MessageHandler.Msg.Name:='Service Error';
		MessageHandler.Msg.Text:=CONCAT(MessageHandler.Msg.Text,ErrorMsg);
		MessageHandler.Msg.Station:=0;

		MessageHandler(
			Prio:=2, 							(*1=highest, .. , 4=lowest*)
			Btn1Addr:=ADR(MsgOk),	(*Address of Button1 , if Zero then Button is unvisible*)
			Btn2Addr:=,						(*Address of Button2 , if Zero then Button is unvisible*)
			sVisu:=Visu.Message);
			(*-----------------------Weiterschaltbedingungen----------------------------*)
		IF MsgOK THEN
				MsgOk:=FALSE;
				ErrorMsg:='';
				fb_state_entry.i16_next_step:=0;
		END_IF

		Error := TRUE;

(*=======================================================*)
	STOP:
		IF fb_state_entry.E THEN
			MessageHandler.ClearMessageLines(sVisu:=Visu.Message);
		END_IF
		(* WARNUNG *)
		MessageHandler.Msg.ID:=ErrorID;
		MessageHandler.Msg.Color:=Color.yellow;
		MessageHandler.Msg.Name:='Service Warnung';
		MessageHandler.Msg.Text:=CONCAT(MessageHandler.Msg.Text,ErrorMsg);
		MessageHandler.Msg.Station:=0;


		MessageHandler(
			Prio:=2, 							(*1=highest, .. , 4=lowest*)
			Btn1Addr:=ADR(MsgOk),	(*Address of Button1 , if Zero then Button is unvisible*)
			Btn2Addr:=,						(*Address of Button2 , if Zero then Button is unvisible*)
			sVisu:=Visu.Message);
			(*-----------------------Weiterschaltbedingungen----------------------------*)
		IF MsgOK THEN
				MsgOk:=FALSE;
				ErrorMsg:='';
				fb_state_entry.i16_next_step:=0;
		END_IF

END_CASE

fb_state_entry(i16_pos:= 2);

fb_bbgen_xml_file(
	start_lesen_service:= ,
	start_schreiben_service:= ,
	s_path:= ,
	s_service:= ,
	fertig_lesen=> ,
	fertig_schreiben=> ,
	bError=> ,
	nErrId=> );


fb_ExpActService(
	Start:= ,
	ExportStr:=CONCAT(CURRENTLANGUAGE,'_Service.xml') ,
	FileName:= 'ActService.txt',
	Path:=  s_tools_path,
	Mode:=FOPEN_MODEWRITE,
	Busy=> ,
	Done=> ,
	Error=> ,
	ErrorMsg=> );
END_PROGRAM
ACTION Button_Init:
(*=====================================================================*)
FOR i:=0 TO 15 BY 1 DO
	Service.visu[i].BtnReset.Text := 'Reset';
	Service.visu[i].BtnReset.Enable := TRUE;
	Service.visu[i].BtnReset.BackgroundColor := Color.lightgrey;
	Service.visu[i].BtnReset.TextColor := Color.black;
	Service.visu[i].BtnReset.Visible := TRUE;


(*=====================================================================*)

	Service.visu[i].BtnStart.Text := 'Start';
	Service.visu[i].BtnStart.Enable := TRUE;
	Service.visu[i].BtnStart.BackgroundColor := Color.lightgrey;
	Service.visu[i].BtnStart.TextColor := Color.black;
	Service.visu[i].BtnStart.Visible := TRUE;


(*=====================================================================*)
	IF 	Service.daten[i].Type_Service = STUNDEN THEN
		Service.visu[i].BtnType.Text := 'TIMER';
		Service.visu[i].BtnType.Pressed := FALSE;
	ELSIF 	Service.daten[i].Type_Service = TAGE THEN
		Service.visu[i].BtnType.Text := 'TIMER';
		Service.visu[i].BtnType.Pressed := FALSE;
	ELSIF Service.daten[i].Type_Service = COUNTER THEN
		Service.visu[i].BtnType.Text := 'COUNT';
		Service.visu[i].BtnType.Pressed := TRUE;
	END_IF
	Service.visu[i].BtnType.Enable := TRUE;
	Service.visu[i].BtnType.BackgroundColor := Color.lightgrey;
	Service.visu[i].BtnType.TextColor := Color.black;
	Service.visu[i].BtnType.Visible := TRUE;
END_FOR
END_ACTION
ACTION Reset:
k:=-1;
FOR k:=1 TO 3 BY 1 DO
	IF	gVarSystemtime.wHour >(MP.ShiftData.Shift[k].TimeStart.wHour + 1) AND NOT Reset_Help[k] THEN
		i:=-1;
		FOR i:=0 TO 15 BY 1 DO
			Default_reached[i] := FALSE;
		END_FOR
		Reset_Help[k]:=TRUE;
	END_IF
END_FOR

IF	gVarSystemtime.wHour < MP.ShiftData.Shift[1].TimeStart.wHour THEN
	k:=-1;
	FOR k:=1 TO 3 BY 1 DO
		Reset_Help[k]:=FALSE;
	END_FOR
END_IF
END_ACTION
ACTION Umschalten:
i := -1;

FOR i:=0 TO 15 BY 1 DO

(* Umschaltung der Funktion (Zeit oder Stückzahl) *)
	IF NOT b_first_cycle THEN
		IF	M_BtnType[i] AND NOT Service.visu[i].BtnType.Pressed THEN
				Service.daten[i].Starttag := 0;
				Service.daten[i].Startstunden := 0;
				Service.daten[i].StartBetriebsStd := 0;
				Service.daten[i].Current_Value := 0;
				IF	Service.daten[i].Type_Service < COUNTER THEN
						Service.daten[i].Type_Service:=Service.daten[i].Type_Service+1;
				ELSE
						Service.daten[i].Type_Service:=0;
				END_IF
		END_IF
		M_BtnType[i]:=Service.visu[i].BtnType.Pressed;

		IF	Service.daten[i].Type_Service = BETRIEBSSTUNDEN THEN
				Service.visu[i].BtnType.Text := 'TIMER';
				Service.daten[i].Unit := 'Betrieb Std';
		END_IF
		IF	Service.daten[i].Type_Service = STUNDEN THEN
				Service.visu[i].BtnType.Text := 'TIMER';
				Service.daten[i].Unit := 'Std';
		END_IF
		IF	Service.daten[i].Type_Service = TAGE THEN
				Service.visu[i].BtnType.Text := 'TIMER';
				Service.daten[i].Unit := 'Tage';
		END_IF
		IF	Service.daten[i].Type_Service = COUNTER THEN
				Service.visu[i].BtnType.Text := 'COUNT';
				Service.daten[i].Unit := 'Zähler';
		END_IF

	END_IF

	(*nur ganze Werte elauben*)
	IF	Service.daten[i].Type_Service = COUNTER OR
			Service.daten[i].Type_Service = TAGE THEN
			HelpString:=LREAL_TO_FMTSTR(Service.daten[i].Default_Value,0,TRUE);
			Service.daten[i].Default_Value:=STRING_TO_LREAL(HelpString);

			HelpString:=LREAL_TO_FMTSTR(Service.daten[i].Warning_Value,0,TRUE);
			Service.daten[i].Warning_Value:=STRING_TO_LREAL(HelpString);
	END_IF
	(* Werte auf 2 Stellen nach dem Komma begrenzen begrenzen*)
	IF	Service.daten[i].Type_Service = STUNDEN OR
			Service.daten[i].Type_Service = BETRIEBSSTUNDEN THEN
			HelpString:=LREAL_TO_FMTSTR(Service.daten[i].Default_Value,2,TRUE);
			Service.daten[i].Default_Value:=STRING_TO_LREAL(HelpString);

			HelpString:=LREAL_TO_FMTSTR(Service.daten[i].Warning_Value,2,TRUE);
			Service.daten[i].Warning_Value:=STRING_TO_LREAL(HelpString);
	END_IF

	(* aktuellen Werte löschen wenn Vorgabe und Warngrenze auf 0 steht*)
	IF	Service.daten[i].Warning_Value=0 AND Service.daten[i].Default_Value=0 THEN
			Service.daten[i].Current_Value:=0;
			Service.visu[i].Current_Value := '0';
			Service.daten[i].Starttag := 0;
			Service.daten[i].Startstunden := 0;
			Service.daten[i].StartBetriebsStd := 0;
			Service.daten[i].Current_Value := 0;
	END_IF

	(*======================================================================================================*)
	CASE Service.daten[i].Type_Service OF

	BETRIEBSSTUNDEN:
			(* Vorgabe erreicht Timer BETRIEBSSTUNDEN  *)
			IF	lr_Betriebsstunden - Service.daten[i].Default_Value >= Service.daten[i].StartBetriebsStd AND
					Service.daten[i].Default_Value >0 AND Service.daten[i].Startstunden >0 THEN
					Service.daten[i].Default_reached := TRUE;
			ELSE
					Service.daten[i].Default_reached := FALSE;
			END_IF

			(* Warngrenze erreicht Timer BETRIEBSSTUNDEN  *)
			IF	lr_Betriebsstunden - Service.daten[i].Warning_Value >= Service.daten[i].StartBetriebsStd AND
					Service.daten[i].Warning_Value >0 AND Service.daten[i].Startstunden >0 THEN
					Service.daten[i].Warning_reached := TRUE;
			ELSE
				Service.daten[i].Warning_reached := FALSE;
			END_IF

		(* Aktuellen Wert  auf der Visu anzeigen *)
		IF Service.daten[i].Starttag >0 THEN
			Service.visu[i].Current_Value :=LREAL_TO_FMTSTR(lr_Betriebsstunden - Service.daten[i].StartBetriebsStd,2,TRUE);
		ELSE
			Service.visu[i].Current_Value := '0';
		END_IF

		(* Start Button für BETRIEBSSTUNDEN sichtbar machen und bei betätigen den aktuellen Tag abspeichern *)
		IF 	Service.daten[i].Starttag =0 AND Service.daten[i].Default_Value >0 THEN
				Service.visu[i].BtnStart.Visible := TRUE;
				IF Service.visu[i].BtnStart.Pressed THEN
					Service.daten[i].Starttag := i_aktueller_tag;
					Service.daten[i].Startstunden := lr_aktuelle_stunden;
					Service.daten[i].StartBetriebsStd := lr_Betriebsstunden;
				END_IF
		ELSE
			Service.visu[i].BtnStart.Visible := FALSE;
		END_IF

	(*======================================================================================================*)
	STUNDEN:
			(* Vorgabe erreicht Timer STUNDEN  *)
			IF	(i_aktueller_tag * 24 + lr_aktuelle_stunden) - (Service.daten[i].Starttag * 24 + Service.daten[i].Startstunden) >= Service.daten[i].Default_Value AND
					Service.daten[i].Default_Value >0 AND Service.daten[i].Startstunden >0 THEN
					Service.daten[i].Default_reached := TRUE;
			ELSE
					Service.daten[i].Default_reached := FALSE;
			END_IF

			(* Warngrenze erreicht Timer STUNDEN  *)
			IF	(i_aktueller_tag * 24 + lr_aktuelle_stunden) - (Service.daten[i].Starttag * 24 + Service.daten[i].Startstunden) >= Service.daten[i].Warning_Value AND
					Service.daten[i].Warning_Value >0 AND Service.daten[i].Startstunden >0 THEN
					Service.daten[i].Warning_reached := TRUE;
			ELSE
				Service.daten[i].Warning_reached := FALSE;
			END_IF

		(* Aktuellen Wert  auf der Visu anzeigen *)
		IF Service.daten[i].Starttag >0 THEN
			Service.visu[i].Current_Value :=LREAL_TO_FMTSTR((i_aktueller_tag * 24 + lr_aktuelle_stunden) - (Service.daten[i].Starttag * 24 + Service.daten[i].Startstunden),2,TRUE);
		ELSE
			Service.visu[i].Current_Value := '0';
		END_IF

		(* Start Button für STUNDEN sichtbar machen und bei betätigen den aktuellen Tag abspeichern *)
		IF  Service.daten[i].Starttag =0 AND Service.daten[i].Default_Value >0 THEN
				Service.visu[i].BtnStart.Visible := TRUE;
				IF Service.visu[i].BtnStart.Pressed THEN
					Service.daten[i].Starttag := i_aktueller_tag;
					Service.daten[i].Startstunden := lr_aktuelle_stunden;
					Service.daten[i].StartBetriebsStd := lr_Betriebsstunden;
				END_IF
		ELSE
			Service.visu[i].BtnStart.Visible := FALSE;
		END_IF

	(*======================================================================================================*)
	TAGE:
		(* Vorgabe erreicht Timer TAGE*)
		IF (i_aktueller_tag - Service.daten[i].Starttag) >= Service.daten[i].Default_Value AND Service.daten[i].Default_Value >0 AND Service.daten[i].Starttag >0 THEN
			Service.daten[i].Default_reached := TRUE;
		ELSE
			Service.daten[i].Default_reached := FALSE;
		END_IF
		(* Warngrenze erreicht Timer TAGE  *)
		IF (i_aktueller_tag - Service.daten[i].Starttag) >= Service.daten[i].Warning_Value AND Service.daten[i].Warning_Value >0 AND Service.daten[i].Starttag >0 THEN
			Service.daten[i].Warning_reached := TRUE;
		ELSE
			Service.daten[i].Warning_reached := FALSE;
		END_IF

		(* Aktuellen Wert  auf der Visu anzeigen *)
		IF Service.daten[i].Starttag >0 THEN
			Service.visu[i].Current_Value := INT_TO_STRING (i_aktueller_tag - Service.daten[i].Starttag);
		ELSE
			Service.visu[i].Current_Value := '0';
		END_IF

		(* Start Button für TAGE sichtbar machen und bei betätigen den aktuellen Tag abspeichern *)
		IF  Service.daten[i].Starttag =0 AND Service.daten[i].Default_Value >0 THEN
				Service.visu[i].BtnStart.Visible := TRUE;
				IF Service.visu[i].BtnStart.Pressed THEN
					Service.daten[i].Starttag := i_aktueller_tag;
					Service.daten[i].Startstunden := lr_aktuelle_stunden;
					Service.daten[i].StartBetriebsStd := lr_Betriebsstunden;
				END_IF
		ELSE
			Service.visu[i].BtnStart.Visible := FALSE;
		END_IF

	(*======================================================================================================*)
	COUNTER:
	(* Vorgabe erreicht COUNTER*)
		IF Service.daten[i].Current_Value >= Service.daten[i].Default_Value AND Service.daten[i].Default_Value > 0 THEN
			Service.daten[i].Default_reached := TRUE;
		ELSE
			Service.daten[i].Default_reached := FALSE;
		END_IF
		(* Warngrenze erreicht COUNTER *)
		IF Service.daten[i].Current_Value >= Service.daten[i].Warning_Value AND Service.daten[i].Warning_Value > 0 THEN
			Service.daten[i].Warning_reached := TRUE;
		ELSE
			Service.daten[i].Warning_reached := FALSE;
		END_IF

	(* Aktuellen Wert  auf der Visu anzeigen *)
		Service.visu[i].Current_Value := LREAL_TO_FMTSTR(Service.daten[i].Current_Value, 0, TRUE);

		Service.visu[i].BtnStart.Visible := FALSE;
	END_CASE
	(*======================================================================================================*)

	(* Aktuellen Zähler reseten wenn dieser voll ist *)
	IF Service.daten[i].Default_reached OR Service.daten[i].Warning_reached THEN
		Service.visu[i].BtnReset.Visible := TRUE;	(* Den Resettaster nur anzeigen wenn Zähler>Vorgabe oder Zähler>Warnung *)
		IF Service.visu[i].BtnReset.Pressed THEN
			Service.daten[i].Starttag := 0;
			Service.daten[i].Startstunden := 0;
			Service.daten[i].StartBetriebsStd := 0;
			Service.daten[i].Current_Value := 0;
			Service.daten[i].Default_reached := FALSE;
			Service.daten[i].Warning_reached := FALSE;
			Default_reached[i]:=FALSE;
			Warning_reached[i]:=FALSE;
		END_IF
	ELSE
		Service.visu[i].BtnReset.Visible := FALSE;
	END_IF

	(* Farbwechsel des aktuellen Wertes *)
	IF Service.daten[i].Default_reached THEN
		Service.visu[i].Current_Value_Color := color.red;
	ELSIF Service.daten[i].Warning_reached AND NOT Service.daten[i].Default_reached THEN
		Service.visu[i].Current_Value_Color := color.yellow;
	ELSE
		Service.visu[i].Current_Value_Color := color.white;
	END_IF

END_FOR
END_ACTION

(* POU zLibrary/ept/Service/ST_BBGenXMLFile, ST *)
FUNCTION_BLOCK ST_BBGenXMLFile
VAR_INPUT
	(* ISK *)
	start_lesen_service						: BOOL;
	start_schreiben_service					: BOOL;

	(* Wo liegen die Dateien *)
	s_path								: STRING(255);

	(* Welche Dateien? *)
	s_service								: STRING(50);
END_VAR
VAR_OUTPUT
	fertig_lesen							: BOOL;
	fertig_schreiben						: BOOL;

	bError								: BOOL;
	nErrId								: UDINT;
END_VAR
VAR
	fb_state_entry							: ST_StateEntry;
	MsgOK								:BOOL;
	fb_ton_quitt							: TON;
	fb_xml_srv_write						: FB_XmlSrvWriteByName;
	fb_xml_srv_read						: FB_XmlSrvReadByName;
	s_file								: STRING(255);
	s_ErrorText							: STRING(255);
	ErrorID								:STRING(20);
END_VAR
fb_ton_quitt(IN:= , PT:= t#50ms, Q=> , ET=> );

(* ======================================Schrittkette======================================== *)
fb_state_entry(
	i16_next_step:= ,
	i16_pos:= 1,
	s_debugtext:= ,
	E=> ,
	X=> ,
	i16_step=> ,
	i16_last_step=> );


CASE fb_state_entry.i16_step OF
(*=======================================================*)
	0:
		bError := FALSE;
		nErrId := 0;

		s_file := '';
		s_ErrorText := '';
		fertig_lesen := FALSE;
		fertig_schreiben := FALSE;

	IF	fb_state_entry.fb_ton_Step.ET > t#10s THEN
		fb_state_entry.i16_next_step := 10;
	END_IF

(*=======================================================*)
	10:	(* Auslesen der Daten aus den XML-Files *)
		(* Daten lesen *)
		IF start_lesen_service THEN
			s_file := CONCAT(s_path, s_service);
			s_file := CONCAT(s_file,'.xml');
			fb_xml_srv_read.sSymName := '.service';
			fb_xml_srv_read.sXPath := '/root/service';
			fb_state_entry.i16_next_step := 100;
		END_IF

		(* Daten schreiben *)
		IF start_schreiben_service THEN
			s_file := CONCAT(s_path, s_service);
			s_file := CONCAT(s_file,'.xml');
			fb_xml_srv_write.sSymName := '.service';
			fb_xml_srv_write.sXPath := '/root/service';
			fb_state_entry.i16_next_step := 200;
		END_IF

(*=======================================================*)
	100:	(* Starte Daten lesen *)
		IF fb_state_entry.E THEN
			fb_xml_srv_read.bExecute := TRUE;
			fb_xml_srv_read.sFilePath := s_file;
		END_IF

		IF fb_xml_srv_read.bBusy THEN
			fb_xml_srv_read.bExecute := FALSE;
			fb_state_entry.i16_next_step := 110;
		END_IF

(*=======================================================*)
	110:	(* Lesevorgang *)
		IF NOT fb_xml_srv_read.bBusy  THEN
			IF NOT fb_xml_srv_read.bError THEN
				fb_state_entry.i16_next_step := 120;
			ELSE	(* Fehler *)
				nErrId := fb_xml_srv_read.nErrId;
				fb_state_entry.i16_next_step := 1000;
				ErrorID:='PM2';
				s_ErrorText:='Fehler beim Lesen der Service.xml Datei';
			END_IF
		END_IF

(*=======================================================*)
	120:	(* Lesevorgang beendet *)
		IF fb_state_entry.E THEN
			fertig_lesen := TRUE;
		END_IF

		IF NOT start_lesen_service THEN
			fb_state_entry.i16_next_step := 0;
		END_IF

(*=======================================================*)
	200:	(* Starte Daten schreiben *)
		IF fb_state_entry.E THEN
			fb_xml_srv_write.bExecute := TRUE;
			fb_xml_srv_write.sFilePath := s_file;
		END_IF

		IF fb_xml_srv_write.bBusy THEN
			fb_xml_srv_write.bExecute := FALSE;
			fb_state_entry.i16_next_step := 210;
		END_IF

(*=======================================================*)
	210:	(* Schreibvorgang *)
		IF NOT fb_xml_srv_write.bBusy  THEN
			IF NOT fb_xml_srv_write.bError THEN
				fb_state_entry.i16_next_step := 220;
			ELSE	(* Fehler *)
				nErrId := fb_xml_srv_write.nErrId;
				fb_state_entry.i16_next_step := 1000;
				s_ErrorText:=CONCAT('Fehler beim Schreiben der ',s_file);
			END_IF
		END_IF

(*=======================================================*)
	220:	(* Schreibvorgang beendet *)
		IF fb_state_entry.E THEN
			fertig_schreiben := TRUE;
		END_IF

		IF NOT start_schreiben_service THEN
			fb_state_entry.i16_next_step := 0;
		END_IF

(*=======================================================*)
	1000: (* Fehler *)
		IF fb_state_entry.E THEN
			MessageHandler.ClearMessageLines(sVisu:=Visu.Message);
		END_IF

		MessageHandler.Msg.ID:=ErrorID;
		MessageHandler.Msg.Color:=Color.red;
		MessageHandler.Msg.Name:='XML Error';
		MessageHandler.Msg.Text:=s_ErrorText;
		MessageHandler.Msg.Station:=0;

		MessageHandler(
			Prio:=2, 							(*1=highest, .. , 4=lowest*)
			Btn1Addr:=ADR(MsgOk),	(*Address of Button1 , if Zero then Button is unvisible*)
			Btn2Addr:=,						(*Address of Button2 , if Zero then Button is unvisible*)
			sVisu:=Visu.Message);

		(*-----------------------Weiterschaltbedingungen----------------------------*)
		IF MsgOK THEN
				MsgOk:=FALSE;
				fb_state_entry.i16_next_step:=0;
		END_IF

END_CASE


fb_state_entry(
	i16_next_step:= ,
	i16_pos:= 2,
	s_debugtext:= ,
	E=> , 
	X=> ,
	i16_step=> ,
	i16_last_step=> );

(* XML *)
fb_xml_srv_read(
	sNetId:= '',
	ePath:= PATH_GENERIC,
	nMode:= XMLSRV_SKIPMISSING,
	sSymName:= ,
	sFilePath:= ,
	sXPath:= ,
	bExecute:= ,
	tTimeout:= t#10s,
	bBusy=> ,
	bError=> ,
	nErrId=> );

fb_xml_srv_write(
	sNetId:= '',
	ePath:= PATH_GENERIC,
	nMode:= XMLSRV_ADDMISSING,
	sSymName:=  ,
	sFilePath:= ,
	sXPath:= ,
	bExecute:= ,
	tTimeout:= t#10s,
	bBusy=> ,
	bError=> ,
	nErrId=> );
END_FUNCTION_BLOCK

(* POU zLibrary/ept/Service/FB_Betriebsstundenzaehler, ST *)
FUNCTION_BLOCK FB_Betriebsstundenzaehler
VAR_INPUT
	Start					: BOOL;
	Reset					: BOOL;
	i32_betriebssekundenzaehler_in	: UDINT;
END_VAR
VAR_OUTPUT
	i32_betriebssekundenzaehler 	: UDINT;
	lr_betriebsstundenzaehler 		: LREAL;
END_VAR
VAR
	b_first_cycle					: BOOL := TRUE;
	fb_ton							: TON;
	t_betriebssekunden_Merker		: TIME := t#0ms;
	fb_r_trig_Reset					: R_TRIG;
	HelpString						: STRING(255);
END_VAR
IF b_first_cycle AND i32_betriebssekundenzaehler_in <>0 THEN
 	i32_betriebssekundenzaehler := i32_betriebssekundenzaehler_in;
	b_first_cycle := FALSE;
END_IF

fb_r_trig_Reset(CLK:=Reset , Q=> );
IF	fb_r_trig_Reset.Q THEN
		i32_betriebssekundenzaehler:=0;
END_IF

(* nach einer bestimmten Zeit speichern *)
IF	fb_ton.ET > t#15m THEN
		Start:=FALSE;
END_IF

IF NOT Start  THEN
	t_betriebssekunden_Merker := t_betriebssekunden_Merker + fb_ton.ET;
END_IF

fb_ton(IN:=Start, PT:= t#24h, Q=> , ET=> );

IF NOT Start THEN
	i32_betriebssekundenzaehler:=i32_betriebssekundenzaehler + (TIME_TO_UDINT(t_betriebssekunden_Merker)/1000);
	t_betriebssekunden_Merker:=t#0ms;
END_IF

lr_betriebsstundenzaehler:=UDINT_TO_LREAL(i32_betriebssekundenzaehler) / 3600;
HelpString:=LREAL_TO_FMTSTR(lr_betriebsstundenzaehler,2,TRUE);
lr_betriebsstundenzaehler:=STRING_TO_LREAL(HelpString);
END_FUNCTION_BLOCK

(* POU Stations/ST_00/ST00_PRGs/ST00_ImpExp_MP, ST *)
PROGRAM ST00_ImpExp_MP
VAR_INPUT
	Start_write				:BOOL;
	Start_read				:BOOL;
	path						:STRING(255);
	filename					:STRING(255);
END_VAR
VAR
	b_init					:BOOL;
	fb_state_entry				:ST_StateEntry;

	fb_xml_srv_read			: FB_XmlSrvReadByName;
	fb_xml_srv_write			: FB_XmlSrvWriteByName;

	fb_rtrig_Start_read			:R_TRIG;
	fb_rtrig_Start_write_to_server:R_TRIG;
	fb_ton_init				:TON;
	fb_ton_wz				:TON;
	fb_ton_uez				:TON;

	bError					: BOOL;
	nErrId					: UDINT;
	s_info					: STRING;
	MsgOK					: BOOL;
	MsgID					:STRING(20);
	MP_Copy				: sMachPara;
END_VAR

VAR_OUTPUT
	Busy					:BOOL;
	Done					:BOOL;
	Error					:BOOL;
	ErrorMsg					:STRING(255);
END_VAR

VAR CONSTANT
	SymName				:STRING:='.MP';
	xPath					:STRING:='/MP';
END_VAR

VAR_IN_OUT

END_VAR
(*======================================================
   PRG: XML Import und Export der MD
 ------------------------------------------------------
   Auth: 		Werner Friedl    						 
   Date: 		25.10.2017   						     
   Rev.: 		1.0	
   Desc:		
	- Maschinen Parameter werden beim Neustart eingelesen
	- bei einer Änderung wird die Änderung automatisch in die xml eingeragen

   Historie:   1.0



 ========================================================*)
fb_ton_init(IN:= TRUE, PT:=t#1500ms , Q=> , ET=> );
IF	NOT b_init AND fb_ton_init.Q THEN
	Start_read := TRUE;
	b_Init:=TRUE;
END_IF

(* ========================================================*)
fb_rtrig_Start_read();
IF	fb_rtrig_Start_read.Q AND
	NOT Start_write THEN
	Start_read:=TRUE;
END_IF

IF 	(MEMCMP(ADR(MP_Copy),ADR(MP),SIZEOF(MP_Copy))<>0)AND (*automatisch speichern im Manualmode*)
     	ModeSelect.Mode <=MODE_MANUAL AND
	NOT Start_read AND
	b_Init THEN
	Start_write := TRUE;
END_IF

(* ========================================================*)
fb_ton_wz(IN:= , PT:=t#3000ms , Q=> , ET=> );
IF	fb_ton_wz.Q THEN
	fb_ton_wz.IN:=FALSE;
	s_info := '';
END_IF

fb_state_entry(i16_pos:= 1);
CASE fb_state_entry.i16_step OF

(*=======================================================*)
INIT_OBJ:
	fb_state_entry.i16_next_step:=INIT;

(*=======================================================*)
INIT: fb_state_entry.s_debugtext:='initialisieren';

	Start_write := FALSE;
	Start_read := FALSE;
	fb_state_entry.i16_next_step:=BEREIT;

(*=======================================================*)
BEREIT:fb_state_entry.s_debugtext:='warte auf start';

	IF	Start_read THEN
		fb_state_entry.i16_next_step:=110;
	END_IF

	IF	Start_write THEN
		fb_state_entry.i16_next_step:=200;
	END_IF

	IF fb_state_entry.X THEN
		fb_ton_uez.IN:=FALSE;
		Start_write:=FALSE;
		Start_read:=FALSE;
		Busy:=TRUE;
		Error:=FALSE;
		Done:=FALSE;
		nErrId:=0;
		ErrorMsg:='';
		MsgID:='';
	END_IF

(*=======================================================*)
110: fb_state_entry.s_debugtext:='XML auslesen';

	IF fb_state_entry.E THEN
		(*MD:=MD_leer;*)
		fb_xml_srv_read.sFilePath := CONCAT(path,filename);
		fb_xml_srv_read.sSymName:=SymName;
		fb_xml_srv_read.sXPath :=xPath;
		fb_xml_srv_read.bExecute := TRUE;
	END_IF

	IF fb_xml_srv_read.bBusy THEN
		fb_xml_srv_read.bExecute := FALSE;
		fb_state_entry.i16_next_step := 120;
	END_IF

(*=======================================================*)
120:fb_state_entry.s_debugtext:='Lesevorgang erfolgreich?';

	IF  NOT fb_xml_srv_read.bBusy  THEN
		IF NOT fb_xml_srv_read.bError THEN
			fb_state_entry.i16_next_step := 900;
		ELSE	(* Fehler *)
			nErrId := fb_xml_srv_read.nErrId;
			IF	nErrId =1804 THEN
				MsgID:='PM5';
				ErrorMsg:='Die Datei MP.xml ist nicht vorhanden';
				fb_state_entry.i16_next_step := 200;	(*Datei wird erstellt*)
			ELSE
				MsgID:='PM6';
				ErrorMsg:='Fehler beim Einlesen der MP.xml Datei';
				fb_state_entry.i16_next_step := FEHLER;
			END_IF
		END_IF
	END_IF

	IF fb_state_entry.X THEN
		fb_ton_wz.IN:=TRUE;
		s_info:=CONCAT('read ',filename);
	END_IF

(*=======================================================*)
200:fb_state_entry.s_debugtext:='XML schreiben';

	IF fb_state_entry.E THEN
		fb_xml_srv_write.sFilePath := CONCAT(path,filename);
		fb_xml_srv_write.sSymName:=SymName;
		fb_xml_srv_write.sXPath :=xPath;
		fb_xml_srv_write.bExecute := TRUE;
	END_IF

	IF fb_xml_srv_write.bBusy THEN
		fb_xml_srv_write.bExecute := FALSE;
		fb_state_entry.i16_next_step := 220;
	END_IF

(*=======================================================*)
220:fb_state_entry.s_debugtext:='Schreiben erfolgreich?';

	IF  NOT fb_xml_srv_write.bBusy  THEN
		IF NOT fb_xml_srv_write.bError THEN
			MP_Copy := MP;
			fb_state_entry.i16_next_step := 900;
		ELSE	(* Fehler *)
			nErrId := fb_xml_srv_write.nErrId;
			MsgID:='PM7';
			ErrorMsg:='Fehler beim Schreiben der MP.xml';
			fb_state_entry.i16_next_step := FEHLER;
		END_IF
	END_IF

	IF fb_state_entry.X THEN
		fb_ton_wz.IN:=TRUE;
		fb_ton_uez.IN:=TRUE;		(*automatisch auf Server speichern*)
		s_info:=CONCAT('write ',filename);
	END_IF

(*=======================================================*)
900:fb_state_entry.s_debugtext:='Fertig';

	Busy:=FALSE;
	Done:=TRUE;
	fb_state_entry.i16_next_step:=0;

(*=======================================================*)
FEHLER:

	IF fb_state_entry.E THEN
		MessageHandler.ClearMessageLines(sVisu:=Visu.Message);
	END_IF
	MessageHandler.Msg.ID:=MsgID;
	MessageHandler.Msg.Name:=ErrorMsg;
	MessageHandler.Msg.Text:=ErrorMsg;
	MessageHandler.Msg.Color:=Color.red;
	MessageHandler.Msg.Station:=0;

	MessageHandler(
		Prio:=2, 							(*1=highest, .. , 4=lowest*)
		Btn1Addr:=ADR(MsgOk),			(*Address of Button1 , if Zero then Button is unvisible*)
		Btn2Addr:=,						(*Address of Button2 , if Zero then Button is unvisible*)
		sVisu:=Visu.Message);

	IF MsgOK THEN
		MsgOk:=FALSE;
		fb_state_entry.i16_next_step:=0;
		Busy:=FALSE;
		Error:=TRUE;
	END_IF
END_CASE

fb_state_entry(i16_pos:= 2);


fb_xml_srv_read(
	sNetId:= '',
	ePath:= PATH_GENERIC,
	nMode:= XMLSRV_SKIPMISSING,
	sSymName:= ,
	sFilePath:= ,
	sXPath:= ,
	bExecute:= ,
	tTimeout:= t#10s,
	bBusy=> ,
	bError=> ,
	nErrId=> );

fb_xml_srv_write(
	sNetId:= '',
	ePath:= PATH_GENERIC,
	nMode:= XMLSRV_ADDMISSING,
	sSymName:=  ,
	sFilePath:= ,
	sXPath:= ,
	bExecute:= ,
	tTimeout:= t#10s,
	bBusy=> ,
	bError=> ,
	nErrId=> );


(*automatisch auf Server speichern=============================================*)
fb_ton_uez(PT:=t#20s);
fb_rtrig_Start_write_to_server(CLK:=fb_ton_uez.Q , Q=> );
(*
NT_StartProcess(
	NETID:='',
	PATHSTR	:='C:\Windows\System32\cmd.exe',
	DIRNAME	:='D:\Tools ',
	COMNDLINE	:='/C copy C:\MP\MachPara.xml \\10.16.50.9\bbgen\UML3\MD & @ping localhost -n 4 >NUL',
	START		:=fb_rtrig_Start_write_to_server.Q,
	TMOUT		:=t#10s);
*)
(*
NT_StartProcess(
	NETID:='',
	PATHSTR	:='C:\Windows\System32\wscript.exe',
	DIRNAME	:='D:\Tools',
	COMNDLINE	:='de_PD_aktuell_von_uml_nach_server.vbs',
	START		:=fb_rtrig_Start_write_to_server.Q,
	TMOUT		:=t#10s);
*)
END_PROGRAM

(* POU Stations/ST_02_RT_Tampondrucker/ST02_PRGs/ST02_CallPRGs, ST *)
PROGRAM ST02_CallPRGs

VAR
	FB_ReadXmlLineConf		: FB_ReadXmlLine;
	sDescription			: STRING;
END_VAR
TurnTable();

IF 	ST02_HomePosition.State = STATE_RUN THEN
	ListHomeNOK(InstName:='ST02 ',Description:=sDescription);
END_IF
FB_ReadXmlLineConf(
	Prefix:= 'CONFIG',
	ID:= 'ST02',
	File:= 'CONFIG.xml',
	Text=> sDescription );

(*Hauptluft Tampondrucker einschalten*)
IF 	ST08_210_S2.BitInToCheck THEN	(*   Not-Aus 2 TD ausgelöst (DigIn) *)
	ST02_35Y01.MoveWork:=TRUE;
ELSE
	ST02_35Y01.MoveInit:=TRUE;
END_IF
END_PROGRAM

(* POU Stations/ST_02_RT_Tampondrucker/ST02_PRGs/TurnTable, ST *)
PROGRAM TurnTable
VAR_OUTPUT
	TurnEnable				: BOOL;
	TurnDisableString		: STRING(255);
END_VAR
VAR
	Test					: BOOL;
	TurnImp					: R_TRIG;

	TimeOutError			: BOOL;
	NestIdx					: DINT;
END_VAR
(*Interlocking for Turn-Table (used in Manual- and in AutoMode)
  ----------------------------------------------------------------------------------------*)

IF 	Robot01.ActualArea=3 THEN	(*Belade-Roboter bei Rundtisch*)
	TurnEnable:=FALSE;
	TurnDisableString:='Robot01.ActualArea=3 in Rundtisch';
ELSIF
	TimeOutError THEN			(*TimeOutError*)
	TurnEnable:=FALSE;
	TurnDisableString:='TimeOutError';
ELSIF
	ST00_220_S1.BitInToCheck THEN (* Schutz nicht geschlossen*)
	TurnEnable:=FALSE;
	TurnDisableString:='Schutztüre nicht geschlossen! ()';
ELSE
	TurnEnable:=TRUE;
	TurnDisableString:='';
END_IF

(*Daten schieben, wenn Rundtisch dreht
	  ----------------------------------------------------------------------------------------*)
IF ModeSelect.Mode=MODE_MANUAL THEN
	TurnImp(CLK:=		(*ST02_162_A1_3.BitOutToSet OR *)  (*Drehen*)
				Test);
	IF TurnImp.Q THEN
		MP.ST02.TableData:=PushData(MP.ST02.TableData);
	END_IF
END_IF
(*Calculate Table Empty*)
gTableEmpty:=TRUE;
FOR NestIdx:=1 TO NO_OF_NEST DO
	IF 	MP.ST02.TableData[NestIdx].ProcessData.Part THEN
		gTableEmpty:=FALSE;
		EXIT;
	END_IF
END_FOR
END_PROGRAM

(* POU Stations/ST_03_Ruestsaetze/ST_03_PRGs/ST03_CallPRGs, ST *)
PROGRAM ST03_CallPRGs
VAR
	fbTon_EndTestParts    	: TON;
	fb_rTrig_EndTestParts	: R_TRIG;
	fb_rTrig_TestParts 		: R_TRIG;

	FB_ReadXmlLineConf		: FB_ReadXmlLine;
	sDescription			: STRING;
	i						:INT;
 	ST03_Ruestsatz			: ARRAY[1..3] OF SFCCurrent;	(*für Grundstellungs Info*)
 	ST03_RuestsatzEmpty		: ARRAY[1..3] OF SFCCurrent;

END_VAR
ST03_ManRobotSwivelUnit();
ST03_Band();
ST03_Test_Parts();
ST03_Init_Lockings();
ST03_Init_AbholPos();

IF 	ST02_HomePosition.State = STATE_RUN THEN
	ListHomeNOK(InstName:='ST03 ',Description:=sDescription);
END_IF

FB_ReadXmlLineConf(
	Prefix:= 'CONFIG',
	ID:= 'ST03',
	File:= 'CONFIG.xml',
	Text=> sDescription );

(*Clear GipperState, if Gripper is opened*)
IF	 Robot01.RemInToolWorkSensor THEN
	gRob01GripState:=PART_NO;
END_IF

ST03_Autostop();

MP.ST03.NoOfTestParts:=MP.ST03.NoOfTestParts - (MP.ST03.NoOfTestParts MOD TD.PartsInRoboGripper);
IF 	MP.ST03.NoOfTestParts < TD.PartsInRoboGripper THEN
	MP.ST03.NoOfTestParts:=TD.PartsInRoboGripper;
END_IF

(* Förderband Prüfteile *)
IF 	MP.ST03.BeltMotorCheckPartActive THEN
	fbTon_EndTestParts(IN:=NOT gTakeTestParts,PT:=t#10s);
	fb_rTrig_TestParts(CLK:=
						gTakeTestParts AND
						ModeSelect.Mode>MODE_MANUAL);
	fb_rTrig_EndTestParts(CLK:=
						fbTon_EndTestParts.Q OR
						ModeSelect.Mode=MODE_MANUAL);

	IF 	fb_rTrig_TestParts.Q THEN
		ST03_601V1_A1.SetSignalHigh:=TRUE;
	END_IF
	IF	fb_rTrig_EndTestParts.Q THEN
    	ST03_601V1_A1.SetSignalLow:=TRUE;
	END_IF

END_IF
(* Berechnung aller Schlechtteile*)
i32_total_NOK_parts :=gNokPartsColorCam+gNokPartsWingCam+i32_first_parts;

(*Hauptluft Tintenstrahldrucker einschalten nur bei SG-Maschine 3621*)
IF 	MP.ST03.SGM_3621 THEN
	IF 	ST08_210_S2.BitInToCheck THEN	(*   Not-Aus 2 TD ausgelöst (DigIn) *)
		ST03_Y01.MoveWork:=TRUE;
	ELSE
		ST03_Y01.MoveInit:=TRUE;
	END_IF
END_IF

ST03_Ruestsatz:=ST03_RuestsatzEmpty;

CASE  gTypeCode OF
(*160pol============================================================================*)
322:
	ST03_160pol_Zufuehrung(
		b_Printer_Off:=TRUE,
		SFCCurrentPOU=> ST03_Ruestsatz[1].SFCCurrentPOU,
		SFCCurrentStep=> ST03_Ruestsatz[1].SFCCurrentStep,
		SFCTime=>ST03_Ruestsatz[1].SFCTime );
	ST03_160pol_Zufuehrung.FB_CurrentStepHistorie(st_CurrentStep:=ST03_160pol_Zufuehrung.SFCCurrentStep);

	IF	(ModeSelect.Mode=MODE_AUTO_RUN OR 	ModeSelect.Mode=MODE_STEP_RUN) AND
		NOT gRunEmpty THEN
		ST03_160pol_Zufuehrung.Start:=TRUE;
	ELSE
		ST03_160pol_Zufuehrung.Start:=FALSE;
	END_IF

(*154pol=============================================================================*)
4871:
	ST03_154pol_Zufuehrung(
		SFCCurrentPOU=> ST03_Ruestsatz[1].SFCCurrentPOU,
		SFCCurrentStep=> ST03_Ruestsatz[1].SFCCurrentStep,
		SFCTime=>ST03_Ruestsatz[1].SFCTime );
	ST03_154pol_Zufuehrung.FB_CurrentStepHistorie(st_CurrentStep:=ST03_154pol_Zufuehrung.SFCCurrentStep);

	IF	(ModeSelect.Mode=MODE_AUTO_RUN OR 	ModeSelect.Mode=MODE_STEP_RUN)	AND
		NOT gRunEmpty THEN
		ST03_154pol_Zufuehrung.Start:=TRUE;
	ELSE
		ST03_154pol_Zufuehrung.Start:=FALSE;
	END_IF

(*154 Rasterplatte=============================================================================*)
4872:
	ST03_154_RP_Zufuehrung(
		SFCCurrentPOU=> ST03_Ruestsatz[1].SFCCurrentPOU,
		SFCCurrentStep=> ST03_Ruestsatz[1].SFCCurrentStep,
		SFCTime=>ST03_Ruestsatz[1].SFCTime );
	ST03_154_RP_Zufuehrung.FB_CurrentStepHistorie(st_CurrentStep:=ST03_154_RP_Zufuehrung.SFCCurrentStep);

	IF	(ModeSelect.Mode=MODE_AUTO_RUN OR 	ModeSelect.Mode=MODE_STEP_RUN)	AND
		NOT gRunEmpty THEN
		ST03_154_RP_Zufuehrung.Start:=TRUE;
	ELSE
		ST03_154_RP_Zufuehrung.Start:=FALSE;
	END_IF

(*93pol, 102pol=============================================================================*)
312,4991:
	ST03_102pol_Zufuehrung(
		SFCCurrentPOU=> ST03_Ruestsatz[1].SFCCurrentPOU,
		SFCCurrentStep=> ST03_Ruestsatz[1].SFCCurrentStep,
		SFCTime=>ST03_Ruestsatz[1].SFCTime );
	ST03_102pol_Zufuehrung.FB_CurrentStepHistorie(st_CurrentStep:=ST03_102pol_Zufuehrung.SFCCurrentStep);

	IF	(ModeSelect.Mode=MODE_AUTO_RUN OR 	ModeSelect.Mode=MODE_STEP_RUN)OR MP.ST02.DummyPruefung_93pol	AND
		NOT gRunEmpty THEN
		ST03_102pol_Zufuehrung.Start:=TRUE;
	ELSE
		ST03_102pol_Zufuehrung.Start:=FALSE;
	END_IF
	IF	MP.ST00.IFMCameraActive THEN
		ST03_IFM_Camera();
		ST03_IFM_Camera.FB_CurrentStepHistorie(st_CurrentStep:=ST03_IFM_Camera.SFCCurrentStep);
	END_IF

(*206pol=============================================================================*)
522:
	ST03_206pol_Zufuehrung(
		SFCCurrentPOU=> ST03_Ruestsatz[1].SFCCurrentPOU,
		SFCCurrentStep=> ST03_Ruestsatz[1].SFCCurrentStep,
		SFCTime=>ST03_Ruestsatz[1].SFCTime );
	ST03_206pol_Zufuehrung.FB_CurrentStepHistorie(st_CurrentStep:=ST03_206pol_Zufuehrung.SFCCurrentStep);

	IF	(ModeSelect.Mode=MODE_AUTO_RUN OR 	ModeSelect.Mode=MODE_STEP_RUN)	AND
		NOT gRunEmpty THEN
		ST03_206pol_Zufuehrung.Start:=TRUE;
	ELSE
		ST03_206pol_Zufuehrung.Start:=FALSE;
	END_IF

(*92pol=============================================================================*)
550:
	ST03_92pol_Zufuehrung(
		SFCCurrentPOU=> ST03_Ruestsatz[1].SFCCurrentPOU,
		SFCCurrentStep=> ST03_Ruestsatz[1].SFCCurrentStep,
		SFCTime=>ST03_Ruestsatz[1].SFCTime );
	ST03_92pol_Zufuehrung.FB_CurrentStepHistorie(st_CurrentStep:=ST03_92pol_Zufuehrung.SFCCurrentStep);

	IF	(ModeSelect.Mode=MODE_AUTO_RUN OR 	ModeSelect.Mode=MODE_STEP_RUN)	AND
		NOT gRunEmpty THEN
		ST03_92pol_Zufuehrung.Start:=TRUE;
	ELSE
		ST03_92pol_Zufuehrung.Start:=FALSE;
	END_IF

(*124pol=============================================================================*)
564:
	ST03_124pol_Zufuehrung(
		SFCCurrentPOU=> ST03_Ruestsatz[1].SFCCurrentPOU,
		SFCCurrentStep=> ST03_Ruestsatz[1].SFCCurrentStep,
		SFCTime=>ST03_Ruestsatz[1].SFCTime );
	ST03_124pol_Zufuehrung.FB_CurrentStepHistorie(st_CurrentStep:=ST03_124pol_Zufuehrung.SFCCurrentStep);

	IF	(ModeSelect.Mode=MODE_AUTO_RUN OR 	ModeSelect.Mode=MODE_STEP_RUN)	AND
		NOT gRunEmpty THEN
		ST03_124pol_Zufuehrung.Start:=TRUE;
	ELSE
		ST03_124pol_Zufuehrung.Start:=FALSE;
	END_IF

(*46pol=============================================================================*)
569:
	ST03_46pol_Zufuehrung(
		SFCCurrentPOU=> ST03_Ruestsatz[1].SFCCurrentPOU,
		SFCCurrentStep=> ST03_Ruestsatz[1].SFCCurrentStep,
		SFCTime=>ST03_Ruestsatz[1].SFCTime );
	ST03_46pol_Zufuehrung.FB_CurrentStepHistorie(st_CurrentStep:=ST03_46pol_Zufuehrung.SFCCurrentStep);
	ST03_46pol_Wendeeinheit(
		SFCCurrentPOU=> ST03_Ruestsatz[2].SFCCurrentPOU,
		SFCCurrentStep=> ST03_Ruestsatz[2].SFCCurrentStep,
		SFCTime=>ST03_Ruestsatz[2].SFCTime );
	ST03_46pol_Wendeeinheit.FB_CurrentStepHistorie(st_CurrentStep:=ST03_46pol_Wendeeinheit.SFCCurrentStep);


	IF	(ModeSelect.Mode=MODE_AUTO_RUN OR 	ModeSelect.Mode=MODE_STEP_RUN)	AND
		NOT gRunEmpty THEN
		ST03_46pol_Zufuehrung.Start:=TRUE;
		ST03_46pol_Wendeeinheit.Start:=TRUE;
	ELSE
		ST03_46pol_Zufuehrung.Start:=FALSE;
		ST03_46pol_Wendeeinheit.Start:=FALSE;
	END_IF

(*NOX 4pol=============================================================================*)
5631:
	ST03_NOX_4pol_Zufuehrung(
		SFCCurrentPOU=> ST03_Ruestsatz[1].SFCCurrentPOU,
		SFCCurrentStep=> ST03_Ruestsatz[1].SFCCurrentStep,
		SFCTime=>ST03_Ruestsatz[1].SFCTime );
	ST03_NOX_4pol_Zufuehrung.FB_CurrentStepHistorie(st_CurrentStep:=ST03_NOX_4pol_Zufuehrung.SFCCurrentStep);

	IF	(ModeSelect.Mode=MODE_AUTO_RUN OR 	ModeSelect.Mode=MODE_STEP_RUN)	AND
		NOT gRunEmpty THEN
		ST03_NOX_4pol_Zufuehrung.Start:=TRUE;
		ST03_65_Q1.SetSignalHigh := TRUE;		(*Kühltunnel (Lüfter)*)
	ELSE
		ST03_NOX_4pol_Zufuehrung.Start:=FALSE;
		ST03_65_Q1.SetSignalLow := TRUE;		(*Kühltunnel (Lüfter)*)
	END_IF

(*NOX 5pol=============================================================================*)
5632:
	ST03_NOX_5pol_Zufuehrung(
		SFCCurrentPOU=> ST03_Ruestsatz[1].SFCCurrentPOU,
		SFCCurrentStep=> ST03_Ruestsatz[1].SFCCurrentStep,
		SFCTime=>ST03_Ruestsatz[1].SFCTime );
	ST03_NOX_5pol_Zufuehrung.FB_CurrentStepHistorie(st_CurrentStep:=ST03_NOX_5pol_Zufuehrung.SFCCurrentStep);

	IF	(ModeSelect.Mode=MODE_AUTO_RUN OR 	ModeSelect.Mode=MODE_STEP_RUN)	AND
		NOT gRunEmpty THEN
		ST03_NOX_5pol_Zufuehrung.Start:=TRUE;
		ST03_65_Q1.SetSignalHigh := TRUE;		(*Kühltunnel (Lüfter)*)
	ELSE
		ST03_NOX_5pol_Zufuehrung.Start:=FALSE;
		ST03_65_Q1.SetSignalLow := TRUE;		(*Kühltunnel (Lüfter)*)
	END_IF

(*NOX 6pol=============================================================================*)
5633:
	ST03_NOX_6pol_Zufuehrung(
		SFCCurrentPOU=> ST03_Ruestsatz[1].SFCCurrentPOU,
		SFCCurrentStep=> ST03_Ruestsatz[1].SFCCurrentStep,
		SFCTime=>ST03_Ruestsatz[1].SFCTime );
	ST03_NOX_6pol_Zufuehrung.FB_CurrentStepHistorie(st_CurrentStep:=ST03_NOX_6pol_Zufuehrung.SFCCurrentStep);

	IF	(ModeSelect.Mode=MODE_AUTO_RUN OR 	ModeSelect.Mode=MODE_STEP_RUN)	AND
		NOT gRunEmpty THEN
		ST03_NOX_6pol_Zufuehrung.Start:=TRUE;
		ST03_65_Q1.SetSignalHigh := TRUE;		(*Kühltunnel (Lüfter)*)
	ELSE
		ST03_NOX_6pol_Zufuehrung.Start:=FALSE;
		ST03_65_Q1.SetSignalLow := TRUE;		(*Kühltunnel (Lüfter)*)
	END_IF

(*88pol=============================================================================*)
5731:
	ST03_88pol_Zufuehrung(
		SFCCurrentPOU=> ST03_Ruestsatz[1].SFCCurrentPOU,
		SFCCurrentStep=> ST03_Ruestsatz[1].SFCCurrentStep,
		SFCTime=>ST03_Ruestsatz[1].SFCTime );
	ST03_88pol_Zufuehrung.FB_CurrentStepHistorie(st_CurrentStep:=ST03_88pol_Zufuehrung.SFCCurrentStep);

	IF	(ModeSelect.Mode=MODE_AUTO_RUN OR 	ModeSelect.Mode=MODE_STEP_RUN)	AND
		NOT gRunEmpty THEN
		ST03_88pol_Zufuehrung.Start:=TRUE;
	ELSE
		ST03_88pol_Zufuehrung.Start:=FALSE;
	END_IF

(*7pol=============================================================================*)
575,5753,5754:
	ST03_7pol_Zufuehrung(
		SFCCurrentPOU=> ST03_Ruestsatz[1].SFCCurrentPOU,
		SFCCurrentStep=> ST03_Ruestsatz[1].SFCCurrentStep,
		SFCTime=>ST03_Ruestsatz[1].SFCTime );
	ST03_7pol_Zufuehrung.FB_CurrentStepHistorie(st_CurrentStep:=ST03_7pol_Zufuehrung.SFCCurrentStep);
	ST03_7pol_Wendeeinheit(
		SFCCurrentPOU=> ST03_Ruestsatz[2].SFCCurrentPOU,
		SFCCurrentStep=> ST03_Ruestsatz[2].SFCCurrentStep,
		SFCTime=>ST03_Ruestsatz[2].SFCTime );
	ST03_7pol_Wendeeinheit.FB_CurrentStepHistorie(st_CurrentStep:=ST03_7pol_Wendeeinheit.SFCCurrentStep);
	IF	(ModeSelect.Mode=MODE_AUTO_RUN OR 	ModeSelect.Mode=MODE_STEP_RUN)	AND
		NOT gRunEmpty THEN
		ST03_7pol_Zufuehrung.Start:=TRUE;
		ST03_7pol_Wendeeinheit.Start:=TRUE;
	ELSE
		ST03_7pol_Zufuehrung.Start:=FALSE;
		ST03_7pol_Wendeeinheit.Start:=FALSE;
	END_IF

(*9pol=============================================================================*)
5755:
	ST03_7pol_Zufuehrung(
		SFCCurrentPOU=> ST03_Ruestsatz[1].SFCCurrentPOU,
		SFCCurrentStep=> ST03_Ruestsatz[1].SFCCurrentStep,
		SFCTime=>ST03_Ruestsatz[1].SFCTime );
	ST03_7pol_Zufuehrung.FB_CurrentStepHistorie(st_CurrentStep:=ST03_7pol_Zufuehrung.SFCCurrentStep);
	ST03_9pol_Wendeeinheit(
		SFCCurrentPOU=> ST03_Ruestsatz[2].SFCCurrentPOU,
		SFCCurrentStep=> ST03_Ruestsatz[2].SFCCurrentStep,
		SFCTime=>ST03_Ruestsatz[2].SFCTime );
	ST03_9pol_Wendeeinheit.FB_CurrentStepHistorie(st_CurrentStep:=ST03_7pol_Wendeeinheit.SFCCurrentStep);
	IF	(ModeSelect.Mode=MODE_AUTO_RUN OR 	ModeSelect.Mode=MODE_STEP_RUN)	AND
		NOT gRunEmpty THEN
		ST03_7pol_Zufuehrung.Start:=TRUE;
		ST03_9pol_Wendeeinheit.Start:=TRUE;
	ELSE
		ST03_7pol_Zufuehrung.Start:=FALSE;
		ST03_9pol_Wendeeinheit.Start:=FALSE;
	END_IF

(*88pol AMG=============================================================================*)
5732:
	ST03_88polAMG_Zufuehrung(
		SFCCurrentPOU=> ST03_Ruestsatz[1].SFCCurrentPOU,
		SFCCurrentStep=> ST03_Ruestsatz[1].SFCCurrentStep,
		SFCTime=>ST03_Ruestsatz[1].SFCTime );
	ST03_88polAMG_Zufuehrung.FB_CurrentStepHistorie(st_CurrentStep:=ST03_88polAMG_Zufuehrung.SFCCurrentStep);

	IF	(ModeSelect.Mode=MODE_AUTO_RUN OR 	ModeSelect.Mode=MODE_STEP_RUN)	AND
		NOT gRunEmpty THEN
		ST03_88polAMG_Zufuehrung.Start:=TRUE;
	ELSE
		ST03_88polAMG_Zufuehrung.Start:=FALSE;
	END_IF

(*120pol AMG=============================================================================*)
5771:
	ST03_120pol_Zufuehrung(
		SFCCurrentPOU=> ST03_Ruestsatz[1].SFCCurrentPOU,
		SFCCurrentStep=> ST03_Ruestsatz[1].SFCCurrentStep,
		SFCTime=>ST03_Ruestsatz[1].SFCTime );
	ST03_120pol_Zufuehrung.FB_CurrentStepHistorie(st_CurrentStep:=ST03_120pol_Zufuehrung.SFCCurrentStep);

	IF	(ModeSelect.Mode=MODE_AUTO_RUN OR 	ModeSelect.Mode=MODE_STEP_RUN)	AND
		NOT gRunEmpty THEN
		ST03_120pol_Zufuehrung.Start:=TRUE;
	ELSE
		ST03_120pol_Zufuehrung.Start:=FALSE;
	END_IF


(*21pol AMG=============================================================================*)
5772:
	ST03_21pol_Zufuehrung(
		SFCCurrentPOU=> ST03_Ruestsatz[1].SFCCurrentPOU,
		SFCCurrentStep=> ST03_Ruestsatz[1].SFCCurrentStep,
		SFCTime=>ST03_Ruestsatz[1].SFCTime );
	ST03_21pol_Zufuehrung.FB_CurrentStepHistorie(st_CurrentStep:=ST03_21pol_Zufuehrung.SFCCurrentStep);

	IF	(ModeSelect.Mode=MODE_AUTO_RUN OR 	ModeSelect.Mode=MODE_STEP_RUN)	AND
		NOT gRunEmpty THEN
		ST03_21pol_Zufuehrung.Start:=TRUE;
	ELSE
		ST03_21pol_Zufuehrung.Start:=FALSE;
	END_IF

(*191pol =============================================================================*)
580:
	ST03_191pol_Zufuehrung(
		SFCCurrentPOU=> ST03_Ruestsatz[1].SFCCurrentPOU,
		SFCCurrentStep=> ST03_Ruestsatz[1].SFCCurrentStep,
		SFCTime=>ST03_Ruestsatz[1].SFCTime );
	ST03_191pol_Zufuehrung.FB_CurrentStepHistorie(st_CurrentStep:=ST03_191pol_Zufuehrung.SFCCurrentStep);

	IF	(ModeSelect.Mode=MODE_AUTO_RUN OR 	ModeSelect.Mode=MODE_STEP_RUN)	AND
		NOT gRunEmpty THEN
		ST03_191pol_Zufuehrung.Start:=TRUE;
	ELSE
		ST03_191pol_Zufuehrung.Start:=FALSE;
	END_IF

(*72pol =============================================================================*)
5831:
	ST03_72pol_Zufuehrung(
		SFCCurrentPOU=> ST03_Ruestsatz[1].SFCCurrentPOU,
		SFCCurrentStep=> ST03_Ruestsatz[1].SFCCurrentStep,
		SFCTime=>ST03_Ruestsatz[1].SFCTime );
	ST03_72pol_Zufuehrung.FB_CurrentStepHistorie(st_CurrentStep:=ST03_72pol_Zufuehrung.SFCCurrentStep);

	IF	(ModeSelect.Mode=MODE_AUTO_RUN OR 	ModeSelect.Mode=MODE_STEP_RUN)	AND
		NOT gRunEmpty THEN
		ST03_72pol_Zufuehrung.Start:=TRUE;
	ELSE
		ST03_72pol_Zufuehrung.Start:=FALSE;
	END_IF

(*48pol =============================================================================*)
5832:
	ST03_48pol_Zufuehrung(
		SFCCurrentPOU=> ST03_Ruestsatz[1].SFCCurrentPOU,
		SFCCurrentStep=> ST03_Ruestsatz[1].SFCCurrentStep,
		SFCTime=>ST03_Ruestsatz[1].SFCTime );
	ST03_48pol_Zufuehrung.FB_CurrentStepHistorie(st_CurrentStep:=ST03_48pol_Zufuehrung.SFCCurrentStep);

	IF	(ModeSelect.Mode=MODE_AUTO_RUN OR 	ModeSelect.Mode=MODE_STEP_RUN)	AND
		NOT gRunEmpty THEN
		ST03_48pol_Zufuehrung.Start:=TRUE;
	ELSE
		ST03_48pol_Zufuehrung.Start:=FALSE;
	END_IF

(*268pol =============================================================================*)
5841:
	ST03_268pol_Zufuehrung(
		SFCCurrentPOU=> ST03_Ruestsatz[1].SFCCurrentPOU,
		SFCCurrentStep=> ST03_Ruestsatz[1].SFCCurrentStep,
		SFCTime=>ST03_Ruestsatz[1].SFCTime );
	ST03_268pol_Zufuehrung.FB_CurrentStepHistorie(st_CurrentStep:=ST03_268pol_Zufuehrung.SFCCurrentStep);

	IF	(ModeSelect.Mode=MODE_AUTO_RUN OR 	ModeSelect.Mode=MODE_STEP_RUN)	AND
		NOT gRunEmpty THEN
		ST03_268pol_Zufuehrung.Start:=TRUE;
	ELSE
		ST03_268pol_Zufuehrung.Start:=FALSE;
	END_IF

(*102pol neu =============================================================================*)
4993:
	ST03_102pol_neu_Zufuehrung(
		SFCCurrentPOU=> ST03_Ruestsatz[1].SFCCurrentPOU,
		SFCCurrentStep=> ST03_Ruestsatz[1].SFCCurrentStep,
		SFCTime=>ST03_Ruestsatz[1].SFCTime );
	ST03_102pol_neu_Zufuehrung.FB_CurrentStepHistorie(st_CurrentStep:=ST03_102pol_neu_Zufuehrung.SFCCurrentStep);

	IF	(ModeSelect.Mode=MODE_AUTO_RUN OR 	ModeSelect.Mode=MODE_STEP_RUN)	AND
		NOT gRunEmpty THEN
		ST03_102pol_neu_Zufuehrung.Start:=TRUE;
	ELSE
		ST03_102pol_neu_Zufuehrung.Start:=FALSE;
	END_IF


(*268pol RP=============================================================================*)
5842:
	ST03_268_RP_Zufuehrung(
		SFCCurrentPOU=> ST03_Ruestsatz[1].SFCCurrentPOU,
		SFCCurrentStep=> ST03_Ruestsatz[1].SFCCurrentStep,
		SFCTime=>ST03_Ruestsatz[1].SFCTime );
	ST03_268_RP_Zufuehrung.FB_CurrentStepHistorie(st_CurrentStep:=ST03_268_RP_Zufuehrung.SFCCurrentStep);
	ST03_268_RP_Wendeeinheit(
		SFCCurrentPOU=> ST03_Ruestsatz[2].SFCCurrentPOU,
		SFCCurrentStep=> ST03_Ruestsatz[2].SFCCurrentStep,
		SFCTime=>ST03_Ruestsatz[2].SFCTime );
	ST03_268_RP_Wendeeinheit.FB_CurrentStepHistorie(st_CurrentStep:=ST03_268_RP_Wendeeinheit.SFCCurrentStep);
	IF	(ModeSelect.Mode=MODE_AUTO_RUN OR 	ModeSelect.Mode=MODE_STEP_RUN)	AND
		NOT gRunEmpty THEN
		ST03_268_RP_Zufuehrung.Start:=TRUE;
		ST03_268_RP_Wendeeinheit.Start:=TRUE;
	ELSE
		ST03_268_RP_Zufuehrung.Start:=FALSE;
		ST03_268_RP_Wendeeinheit.Start:=FALSE;
	END_IF

(*91pol =============================================================================*)
379:
ST03_91pol_Zufuehrung(
		SFCCurrentPOU=> ST03_Ruestsatz[1].SFCCurrentPOU,
		SFCCurrentStep=> ST03_Ruestsatz[1].SFCCurrentStep,
		SFCTime=>ST03_Ruestsatz[1].SFCTime );
	ST03_91pol_Zufuehrung.FB_CurrentStepHistorie(st_CurrentStep:=ST03_91pol_Zufuehrung.SFCCurrentStep);

	IF	(ModeSelect.Mode=MODE_AUTO_RUN OR 	ModeSelect.Mode=MODE_STEP_RUN)	AND
		NOT gRunEmpty THEN
		ST03_91pol_Zufuehrung.Start:=TRUE;
	ELSE
		ST03_91pol_Zufuehrung.Start:=FALSE;
	END_IF

(*33pol=============================================================================*)
598:
	ST03_33pol_Zufuehrung(
		SFCCurrentPOU=> ST03_Ruestsatz[1].SFCCurrentPOU,
		SFCCurrentStep=> ST03_Ruestsatz[1].SFCCurrentStep,
		SFCTime=>ST03_Ruestsatz[1].SFCTime );
	ST03_33pol_Zufuehrung.FB_CurrentStepHistorie(st_CurrentStep:=ST03_33pol_Zufuehrung.SFCCurrentStep);

	IF	(ModeSelect.Mode=MODE_AUTO_RUN OR 	ModeSelect.Mode=MODE_STEP_RUN)	AND
		NOT gRunEmpty THEN
		ST03_33pol_Zufuehrung.Start:=TRUE;
	ELSE
		ST03_33pol_Zufuehrung.Start:=FALSE;
	END_IF

END_CASE
FOR i:=1 TO 3 BY 1 DO
	ST03_Ruestsatz[i].b_activ:=ST03_Ruestsatz[i].SFCCurrentPOU='-';
END_FOR

(*IFM Kamera=============================================================================*)
IF 	ModeSelect.Mode=MODE_MANUAL THEN
	Visu.ST02_FDB_55X1_7_JOB_BIT1.BitOutToSet:=TD.IFM_CamProgNo.0;
	Visu.ST02_FDB_55X1_7_JOB_BIT2.BitOutToSet:=TD.IFM_CamProgNo.1;

	Visu.ST02_FDB_56X1_7_JOB_BIT1.BitOutToSet:=TD.IFM_CamProgNo.0;
	Visu.ST02_FDB_56X1_7_JOB_BIT2.BitOutToSet:=TD.IFM_CamProgNo.1;
END_IF
END_PROGRAM

(* POU Stations/ST_03_Ruestsaetze/ST_03_PRGs/ST03_ManRobotSwivelUnit, ST *)
PROGRAM ST03_ManRobotSwivelUnit
VAR
 ToggleSwivelOn		: TP;
 ToggleSwivelOff	: TP;
 ToggleBtnOn  		: BOOL;
 ToggleBtnOff  		: BOOL;

END_VAR
ToggleSwivelOn(In:=ToggleBtnOn,Pt:=T#1s);
ToggleSwivelOff(In:=ToggleBtnOff,Pt:=T#1s);

IF 	Robot01.State = STATE_WAIT THEN
 gManSwivelOnRobot01:=ToggleSwivelOn.Q;
 gManSwivelOffRobot01:=ToggleSwivelOff.Q;
END_IF
END_PROGRAM

(* POU Stations/ST_03_Ruestsaetze/ST_03_SFCs/Zufuehrungen/ST03_154pol_Zufuehrung, SFC *)
 PROGRAM ST03_154pol_Zufuehrung
VAR_OUTPUT
	SFCCurrentPOU			: STRING:='ST03_154pol_Zufuehrung';
	SFCCurrentStep			: STRING:='';
	FB_CurrentStepHistorie	: FB_CurrentStepHistorie;
	SFCTime					: DINT;
	State   				: StateObject	:= STATE_WAIT;
	Result  				: StateResult;
END_VAR
VAR_INPUT
	Start					:BOOL;
END_VAR
VAR
	MsgOK				: BOOL;
	MsgCancel			: BOOL;
	SFCRun				: BOOL;
	SFCTimeStart		: TIME;
	Delay				: TON;
	(* Userdefinded area *)

END_VAR
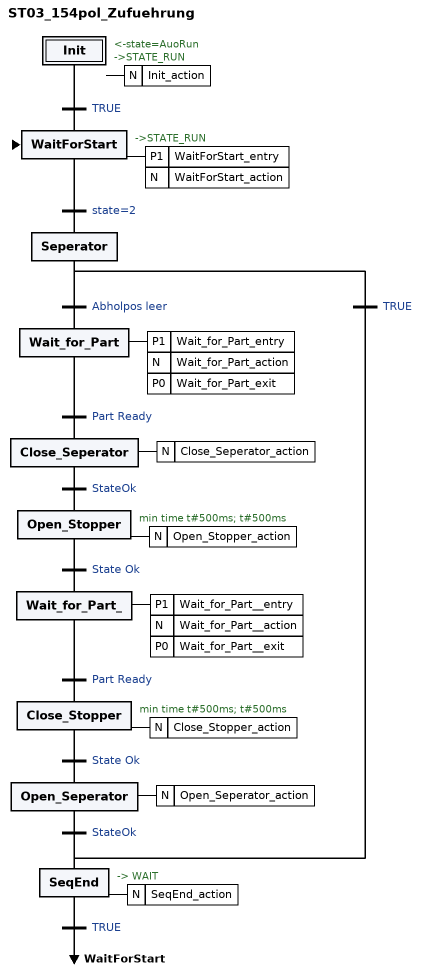
INITIAL_STEP Init: (* <-state=AuoRun / ->STATE_RUN *)
	Init_action(N);
END_STEP
TRANSITION FROM Init TO WaitForStart := TRUE;
END_TRANSITION
STEP WaitForStart: (* ->STATE_RUN *)
	WaitForStart_entry(P1);
	WaitForStart_action(N);
END_STEP
TRANSITION FROM WaitForStart TO Seperator := state=2;
END_TRANSITION
STEP Seperator:
END_STEP
TRANSITION FROM Seperator TO Wait_for_Part := Abholpos leer;
END_TRANSITION
TRANSITION FROM Seperator TO SeqEnd := TRUE;
END_TRANSITION
STEP Wait_for_Part:
	Wait_for_Part_entry(P1);
	Wait_for_Part_action(N);
	Wait_for_Part_exit(P0);
END_STEP
TRANSITION FROM Wait_for_Part TO Close_Seperator := Part Ready;
END_TRANSITION
STEP Close_Seperator:
	Close_Seperator_action(N);
END_STEP
TRANSITION FROM Close_Seperator TO Open_Stopper := StateOk;
END_TRANSITION
STEP Open_Stopper: (* min time t#500ms; t#500ms *)
	Open_Stopper_action(N);
END_STEP
TRANSITION FROM Open_Stopper TO Wait_for_Part_ := State Ok;
END_TRANSITION
STEP Wait_for_Part_:
	Wait_for_Part__entry(P1);
	Wait_for_Part__action(N);
	Wait_for_Part__exit(P0);
END_STEP
TRANSITION FROM Wait_for_Part_ TO Close_Stopper := Part Ready;
END_TRANSITION
STEP Close_Stopper: (* min time t#500ms; t#500ms *)
	Close_Stopper_action(N);
END_STEP
TRANSITION FROM Close_Stopper TO Open_Seperator := State Ok;
END_TRANSITION
STEP Open_Seperator:
	Open_Seperator_action(N);
END_STEP
TRANSITION FROM Open_Seperator TO SeqEnd := StateOk;
END_TRANSITION
STEP SeqEnd: (* -> WAIT *)
	SeqEnd_action(N);
END_STEP
TRANSITION FROM SeqEnd TO WaitForStart := TRUE;
END_TRANSITION

ACTION Init_action:
Start:=FALSE;
State:=STATE_WAIT;
MsgOK:=FALSE;
MsgCancel:=FALSE;
SFCRun:=FALSE;
Result:=RESULT_NON;
END_ACTION

ACTION WaitForStart_entry:
;
END_ACTION

ACTION WaitForStart_action:
IF 	Start   THEN
	State:=STATE_RUN;
	Result:=RESULT_NON;
	SFCTimeStart:=TIME();
	Start:=FALSE;
ELSE
	State:=STATE_WAIT;
	MsgOK:=FALSE;
	MsgCancel:=FALSE;
	SFCRun:=FALSE;
END_IF
END_ACTION

ACTION Wait_for_Part_entry:
ProcessMessage01:='';
Delay.IN:=FALSE;
Delay();
END_ACTION

ACTION Wait_for_Part_action:
ProcessMessage01:='1IM6';(*warte auf Teil in Vereinzelung*)
Delay.IN:=ST03_425_B67_7.BitInToCheck; 		 (* Schnittstelle Iso auf Übergabeposition *)
Delay.PT:=T#500ms;
Delay();
END_ACTION

ACTION Wait_for_Part_exit:
ProcessMessage01:='';
END_ACTION

ACTION Close_Seperator_action:
ST03_426_Y68_5.MoveWork:=TRUE;		(* Förderband  Zuführung Vereinzler AST/GST *)
END_ACTION

ACTION Open_Stopper_action:
ST03_426_Y68_6.MoveWork:=TRUE;		(* Förderband  Züführung Stopper AST/GST *)
END_ACTION

ACTION Wait_for_Part__entry:
ProcessMessage01:='';
Delay.IN:=FALSE;
Delay();
END_ACTION

ACTION Wait_for_Part__action:
ProcessMessage01:='1IM6';(*warte auf Teil in Vereinzelung*)
Delay.IN:=ST03_426_B68_4.BitInToCheck; 		 (* Schnittstelle Iso auf Übergabeposition *)
Delay.PT:=T#500ms;
Delay();
END_ACTION

ACTION Wait_for_Part__exit:
ProcessMessage01:='';
END_ACTION

ACTION Close_Stopper_action:
ST03_426_Y68_6.MoveInit:=TRUE;		(* Förderband  Züführung Stopper AST/GST *)
END_ACTION

ACTION Open_Seperator_action:
ST03_426_Y68_5.MoveInit:=TRUE;		(* Förderband  Zuführung Vereinzler AST/GST *)
END_ACTION

ACTION SeqEnd_action:
SFCTime:=TIME_TO_DINT(TIME()-SFCTimeStart);
State:=STATE_WAIT;
END_ACTION

TRANSITION Abholpos leer:
NOT  ST03_426_B68_4.BitInToCheck
END_TRANSITION

TRANSITION Part Ready:
Delay.Q AND
NOT ST03_426_B68_4.BitInToCheck	AND		(*  Züführung  ISK auf Übergabeposition Roboter Palettierer*)
ST03_425_B67_7.BitInToCheck	AND	(*  ISK anwesend am Vereinzler*)
Robot01.ActualArea <> 4
END_TRANSITION

TRANSITION StateOk:
ST03_426_Y68_5.State=STATE_OK 	(* Förderband  Zuführung Vereinzler AST/GST *)

(*ST03_426_B68_4.BitInToCheck	AND		(*  Züführung  ISK auf Übergabeposition Roboter Palettierer*)
NOT ST03_425_B67_7.BitInToCheck AND	(*  ISK anwesend am Vereinzler*)
gTipImp*)
END_TRANSITION

TRANSITION State Ok:
ST03_426_Y68_6.State=STATE_OK 	(* Förderband  Züführung Stopper AST/GST *)
END_TRANSITION

TRANSITION Part Ready:
Delay.Q AND
(*NOT ST03_426_B68_4.BitInToCheck	AND		(*  Züführung  ISK auf Übergabeposition Roboter Palettierer*)
ST03_425_B67_7.BitInToCheck	AND*)	(*  ISK anwesend am Vereinzler*)
Robot01.ActualArea <> 4
END_TRANSITION

TRANSITION State Ok:
ST03_426_Y68_6.State=STATE_OK 	(* Förderband  Züführung Stopper AST/GST *)
END_TRANSITION

TRANSITION StateOk:
ST03_426_Y68_5.State=STATE_OK 	(* Förderband  Zuführung Vereinzler AST/GST *)

(*ST03_426_B68_4.BitInToCheck	AND		(*  Züführung  ISK auf Übergabeposition Roboter Palettierer*)
NOT ST03_425_B67_7.BitInToCheck AND	(*  ISK anwesend am Vereinzler*)
gTipImp*)
END_TRANSITION
END_PROGRAM

(* POU Stations/ST_03_Ruestsaetze/ST_03_SFCs/Zufuehrungen/ST03_154_RP_Zufuehrung, SFC *)
 PROGRAM ST03_154_RP_Zufuehrung
VAR_OUTPUT
	SFCCurrentPOU			: STRING:='ST03_154_RP_Zufuehrung';
	SFCCurrentStep			: STRING:='';
	FB_CurrentStepHistorie	: FB_CurrentStepHistorie;
	SFCTime					: DINT;
	State   				: StateObject	:= STATE_WAIT;
	Result  				: StateResult;
END_VAR
VAR_INPUT
	Start					:BOOL;
END_VAR
VAR
	MsgOK				: BOOL;
	MsgCancel			: BOOL;
	SFCRun				: BOOL;
	SFCTimeStart		: TIME;
	(* Userdefinded area *)

